LIN {X 0,Y 249.202,Z 538.442,A -85,B 0,C 180,E1 -19004.703,E2 -19004.703} C_VEL
LIN {X 0,Y 249.136,Z 538.448,A -85,B 0,C 180,E1 -19008.077,E2 -19008.077} C_VEL
LIN {X 0,Y 249.084,Z 538.455,A -85,B 0,C 180,E1 -19011.518,E2 -19011.518} C_VEL
LIN {X 0,Y 249.127,Z 538.45,A -85,B 0,C 180,E1 -19015.482,E2 -19015.482} C_VEL
LIN {X 0,Y 249.079,Z 538.459,A -85,B 0,C 180,E1 -19018.993,E2 -19018.993} C_VEL
LIN {X 0,Y 249.032,Z 538.463,A -85,B 0,C 180,E1 -19022.425,E2 -19022.425} C_VEL
LIN {X 0,Y 249.071,Z 538.458,A -85,B 0,C 180,E1 -19026.337,E2 -19026.337} C_VEL
LIN {X 0,Y 249.079,Z 538.453,A -85,B 0,C 180,E1 -19030.463,E2 -19030.463} C_VEL
LIN {X 0,Y 249.089,Z 538.457,A -85,B 0,C 180,E1 -19032.814,E2 -19032.814} C_VEL
LIN {X 0,Y 249.092,Z 538.448,A -85,B 0,C 180,E1 -19037.38,E2 -19037.38} C_VEL
LIN {X 0,Y 249.047,Z 538.461,A -85,B 0,C 180,E1 -19041.624,E2 -19041.624} C_VEL
LIN {X 0,Y 249.055,Z 538.456,A -85,B 0,C 180,E1 -19045.642,E2 -19045.642} C_VEL
LIN {X 0,Y 249.046,Z 538.458,A -85,B 0,C 180,E1 -19049.473,E2 -19049.473} C_VEL
LIN {X 0,Y 249.065,Z 538.462,A -85,B 0,C 180,E1 -19053.162,E2 -19053.162} C_VEL
LIN {X 0,Y 249.055,Z 538.459,A -85,B 0,C 180,E1 -19056.731,E2 -19056.731} C_VEL
LIN {X 0,Y 249.101,Z 538.445,A -85,B 0,C 180,E1 -19060.212,E2 -19060.212} C_VEL
LIN {X 0,Y 249.236,Z 538.437,A -85,B 0,C 180,E1 -19063.622,E2 -19063.622} C_VEL
LIN {X 0,Y 249.247,Z 538.431,A -85,B 0,C 180,E1 -19068.617,E2 -19068.617} C_VEL
LIN {X 0,Y 249.476,Z 538.401,A -85,B 0,C 180,E1 -19071.903,E2 -19071.903} C_VEL
LIN {X 0,Y 249.432,Z 538.412,A -85,B 0,C 180,E1 -19076.77,E2 -19076.77} C_VEL
LIN {X 0,Y 249.73,Z 538.365,A -85,B 0,C 180,E1 -19080.001,E2 -19080.001} C_VEL
LIN {X 0,Y 249.463,Z 538.408,A -85,B 0,C 180,E1 -19083.231,E2 -19083.231} C_VEL
LIN {X 0,Y 249.45,Z 538.405,A -85,B 0,C 180,E1 -19088.099,E2 -19088.099} C_VEL
LIN {X 0,Y 249.218,Z 538.441,A -85,B 0,C 180,E1 -19093.039,E2 -19093.039} C_VEL
LIN {X 0,Y 249.184,Z 538.442,A -85,B 0,C 180,E1 -19094.212,E2 -19094.212} C_VEL
LIN {X 0,Y 248.517,Z 538.528,A -85,B 0,C 180,E1 -19095.561,E2 -19095.561} C_VEL
LIN {X 0,Y 245.6,Z 538.889,A -85,B 0,C 180,E1 -19097.758,E2 -19097.758} C_VEL
LIN {X 0,Y 243.131,Z 539.2,A -85,B 0,C 180,E1 -19099.547,E2 -19099.547} C_VEL
LIN {X 0,Y 242.102,Z 539.328,A -85,B 0,C 180,E1 -19100.938,E2 -19100.938} C_VEL
LIN {X 0,Y 242.035,Z 539.333,A -85,B 0,C 180,E1 -19101.409,E2 -19101.409} C_VEL
LIN {X 0,Y 242.064,Z 539.332,A -85,B 0,C 180,E1 -19105.839,E2 -19105.839} C_VEL
LIN {X 0,Y 242.028,Z 539.335,A -85,B 0,C 180,E1 -19109.581,E2 -19109.581} C_VEL
LIN {X 0,Y 241.989,Z 539.34,A -85,B 0,C 180,E1 -19113.492,E2 -19113.492} C_VEL
LIN {X 0,Y 241.997,Z 539.34,A -85,B 0,C 180,E1 -19117.581,E2 -19117.581} C_VEL
LIN {X 0,Y 241.942,Z 539.347,A -85,B 0,C 180,E1 -19121.922,E2 -19121.922} C_VEL
LIN {X 0,Y 241.991,Z 539.341,A -85,B 0,C 180,E1 -19126.558,E2 -19126.558} C_VEL
LIN {X 0,Y 242.063,Z 539.462,A -85,B 0,C 180,E1 -19131.377,E2 -19131.377} C_VEL
LIN {X 0,Y 244.298,Z 549.492,A -85,B 0,C 180,E1 -19135.282,E2 -19135.282} C_VEL
LIN {X 0,Y 246.378,Z 559.411,A -85,B 0,C 180,E1 -19138.944,E2 -19138.944} C_VEL
LIN {X 0,Y 250.709,Z 571.961,A -85,B 0,C 180,E1 -19139.853,E2 -19139.853} C_VEL
LIN {X 0,Y 255.893,Z 613.107,A -85,B 0,C 180,E1 -19141.765,E2 -19141.765} C_VEL
LIN {X 0,Y 254.09,Z 666.383,A -85,B 0,C 180,E1 -19143.398,E2 -19143.398} C_VEL
LIN {X 0,Y 253.162,Z 679.381,A -85,B 0,C 180,E1 -19144.018,E2 -19144.018} C_VEL
LIN {X 0,Y 251.694,Z 692.993,A -85,B 0,C 180,E1 -19145.019,E2 -19145.019} C_VEL
LIN {X 0,Y 250.086,Z 704.507,A -85,B 0,C 180,E1 -19146.174,E2 -19146.174} C_VEL
LIN {X 0,Y 248.201,Z 716.399,A -85,B 0,C 180,E1 -19147.746,E2 -19147.746} C_VEL
LIN {X 0,Y 246.273,Z 727.047,A -85,B 0,C 180,E1 -19149.539,E2 -19149.539} C_VEL
LIN {X 0,Y 244.509,Z 736.668,A -85,B 0,C 180,E1 -19151.569,E2 -19151.569} C_VEL
LIN {X 0,Y 243.139,Z 744.544,A -85,B 0,C 180,E1 -19153.631,E2 -19153.631} C_VEL
LIN {X 0,Y 241.777,Z 752.217,A -85,B 0,C 180,E1 -19156.125,E2 -19156.125} C_VEL
LIN {X 0,Y 240.683,Z 759.286,A -85,B 0,C 180,E1 -19159.059,E2 -19159.059} C_VEL
LIN {X 0,Y 240.204,Z 763.93,A -85,B 0,C 180,E1 -19161.588,E2 -19161.588} C_VEL
LIN {X 0,Y 240.095,Z 767.755,A -85,B 0,C 180,E1 -19164.414,E2 -19164.414} C_VEL
LIN {X 0,Y 240.067,Z 769.874,A -85,B 0,C 180,E1 -19166.643,E2 -19166.643} C_VEL
LIN {X 0,Y 240.079,Z 770.935,A -85,B 0,C 180,E1 -19168.323,E2 -19168.323} C_VEL
LIN {X 0,Y 240.149,Z 771.574,A -85,B 0,C 180,E1 -19170,E2 -19170} C_VEL
LIN {X 0,Y 240.061,Z 771.798,A -85,B 0,C 180,E1 -19171.678,E2 -19171.678} C_VEL
LIN {X 0,Y 239.982,Z 771.619,A -85,B 0,C 180,E1 -19173.358,E2 -19173.358} C_VEL
LIN {X 0,Y 239.915,Z 770.952,A -85,B 0,C 180,E1 -19175.127,E2 -19175.127} C_VEL
LIN {X 0,Y 240.154,Z 768.543,A -85,B 0,C 180,E1 -19178.414,E2 -19178.414} C_VEL
LIN {X 0,Y 240.703,Z 765.591,A -85,B 0,C 180,E1 -19180.94,E2 -19180.94} C_VEL
LIN {X 0,Y 241.637,Z 761.631,A -85,B 0,C 180,E1 -19183.455,E2 -19183.455} C_VEL
LIN {X 0,Y 243.223,Z 756.564,A -85,B 0,C 180,E1 -19185.932,E2 -19185.932} C_VEL
LIN {X 0,Y 245.134,Z 750.236,A -85,B 0,C 180,E1 -19188.383,E2 -19188.383} C_VEL
LIN {X 0,Y 247.351,Z 742.42,A -85,B 0,C 180,E1 -19190.803,E2 -19190.803} C_VEL
LIN {X 0,Y 250.172,Z 732.673,A -85,B 0,C 180,E1 -19193.159,E2 -19193.159} C_VEL
LIN {X 0,Y 252.937,Z 722.679,A -85,B 0,C 180,E1 -19195.07,E2 -19195.07} C_VEL
LIN {X 0,Y 255.704,Z 711.555,A -85,B 0,C 180,E1 -19196.747,E2 -19196.747} C_VEL
LIN {X 0,Y 258.424,Z 699.033,A -85,B 0,C 180,E1 -19198.198,E2 -19198.198} C_VEL
LIN {X 0,Y 260.641,Z 686.739,A -85,B 0,C 180,E1 -19199.256,E2 -19199.256} C_VEL
LIN {X 0,Y 262.493,Z 673.125,A -85,B 0,C 180,E1 -19200.077,E2 -19200.077} C_VEL
LIN {X 0,Y 263.562,Z 659.455,A -85,B 0,C 180,E1 -19200.616,E2 -19200.616} C_VEL
LIN {X 0,Y 265.646,Z 615.521,A -85,B 0,C 180,E1 -19201.945,E2 -19201.945} C_VEL
LIN {X 0,Y 263.42,Z 595.456,A -85,B 0,C 180,E1 -19203.118,E2 -19203.118} C_VEL
LIN {X 0,Y 261.883,Z 586.129,A -85,B 0,C 180,E1 -19203.783,E2 -19203.783} C_VEL
LIN {X 0,Y 256.187,Z 573.517,A -85,B 0,C 180,E1 -19205.432,E2 -19205.432} C_VEL
LIN {X 0,Y 251.731,Z 564.822,A -85,B 0,C 180,E1 -19206.781,E2 -19206.781} C_VEL
LIN {X 0,Y 249.058,Z 559.92,A -85,B 0,C 180,E1 -19207.624,E2 -19207.624} C_VEL
LIN {X 0,Y 246.628,Z 555.3,A -85,B 0,C 180,E1 -19208.441,E2 -19208.441} C_VEL
LIN {X 0,Y 244.346,Z 546.982,A -85,B 0,C 180,E1 -19212.824,E2 -19212.824} C_VEL
LIN {X 0,Y 242.406,Z 541.046,A -85,B 0,C 180,E1 -19216.452,E2 -19216.452} C_VEL
LIN {X 0,Y 241.976,Z 539.338,A -85,B 0,C 180,E1 -19217.657,E2 -19217.657} C_VEL
LIN {X 0,Y 242,Z 539.336,A -85,B 0,C 180,E1 -19222.419,E2 -19222.419} C_VEL
LIN {X 0,Y 241.989,Z 539.336,A -85,B 0,C 180,E1 -19226.508,E2 -19226.508} C_VEL
LIN {X 0,Y 242.035,Z 539.337,A -85,B 0,C 180,E1 -19230.586,E2 -19230.586} C_VEL
LIN {X 0,Y 242.065,Z 539.333,A -85,B 0,C 180,E1 -19234.182,E2 -19234.182} C_VEL
LIN {X 0,Y 242.05,Z 539.33,A -85,B 0,C 180,E1 -19238.296,E2 -19238.296} C_VEL
LIN {X 0,Y 242.16,Z 539.313,A -85,B 0,C 180,E1 -19243.277,E2 -19243.277} C_VEL
LIN {X 0,Y 242.181,Z 539.318,A -85,B 0,C 180,E1 -19248.279,E2 -19248.279} C_VEL
LIN {X 0,Y 242.422,Z 539.288,A -85,B 0,C 180,E1 -19251.665,E2 -19251.665} C_VEL
LIN {X 0,Y 242.257,Z 539.306,A -85,B 0,C 180,E1 -19255.006,E2 -19255.006} C_VEL
LIN {X 0,Y 242.632,Z 539.26,A -85,B 0,C 180,E1 -19258.339,E2 -19258.339} C_VEL
LIN {X 0,Y 242.634,Z 539.261,A -85,B 0,C 180,E1 -19261.659,E2 -19261.659} C_VEL
LIN {X 0,Y 242.418,Z 539.283,A -85,B 0,C 180,E1 -19266.675,E2 -19266.675} C_VEL
LIN {X 0,Y 242.262,Z 539.308,A -85,B 0,C 180,E1 -19270.023,E2 -19270.023} C_VEL
LIN {X 0,Y 242.181,Z 539.32,A -85,B 0,C 180,E1 -19272.517,E2 -19272.517} C_VEL
LIN {X 0,Y 243.031,Z 541.925,A -85,B 0,C 180,E1 -19272.897,E2 -19272.897} C_VEL
LIN {X 0,Y 244.839,Z 544.043,A -85,B 0,C 180,E1 -19273.486,E2 -19273.486} C_VEL
LIN {X 0,Y 245.625,Z 545.011,A -85,B 0,C 180,E1 -19273.74,E2 -19273.74} C_VEL
LIN {X 0,Y 247.708,Z 548.228,A -85,B 0,C 180,E1 -19274.426,E2 -19274.426} C_VEL
LIN {X 0,Y 249.131,Z 550.181,A -85,B 0,C 180,E1 -19274.864,E2 -19274.864} C_VEL
LIN {X 0,Y 255.936,Z 560.636,A -85,B 0,C 180,E1 -19276.882,E2 -19276.882} C_VEL
LIN {X 0,Y 261.966,Z 571.367,A -85,B 0,C 180,E1 -19278.552,E2 -19278.552} C_VEL
LIN {X 0,Y 266.972,Z 582.249,A -85,B 0,C 180,E1 -19279.921,E2 -19279.921} C_VEL
LIN {X 0,Y 267.197,Z 583.754,A -85,B 0,C 180,E1 -19280.019,E2 -19280.019} C_VEL
LIN {X 0,Y 264.008,Z 643.013,A -85,B 0,C 180,E1 -19281.805,E2 -19281.805} C_VEL
LIN {X 0,Y 262.72,Z 656.866,A -85,B 0,C 180,E1 -19282.537,E2 -19282.537} C_VEL
LIN {X 0,Y 261.055,Z 669.85,A -85,B 0,C 180,E1 -19283.565,E2 -19283.565} C_VEL
LIN {X 0,Y 258.946,Z 682.051,A -85,B 0,C 180,E1 -19284.877,E2 -19284.877} C_VEL
LIN {X 0,Y 256.57,Z 693.258,A -85,B 0,C 180,E1 -19286.43,E2 -19286.43} C_VEL
LIN {X 0,Y 254.034,Z 703.269,A -85,B 0,C 180,E1 -19288.191,E2 -19288.191} C_VEL
LIN {X 0,Y 251.485,Z 712.369,A -85,B 0,C 180,E1 -19290.2,E2 -19290.2} C_VEL
LIN {X 0,Y 248.923,Z 720.553,A -85,B 0,C 180,E1 -19292.441,E2 -19292.441} C_VEL
LIN {X 0,Y 246.775,Z 727.156,A -85,B 0,C 180,E1 -19294.72,E2 -19294.72} C_VEL
LIN {X 0,Y 244.896,Z 732.541,A -85,B 0,C 180,E1 -19297.059,E2 -19297.059} C_VEL
LIN {X 0,Y 243.342,Z 736.838,A -85,B 0,C 180,E1 -19299.447,E2 -19299.447} C_VEL
LIN {X 0,Y 242.128,Z 740.133,A -85,B 0,C 180,E1 -19301.881,E2 -19301.881} C_VEL
LIN {X 0,Y 241.176,Z 742.511,A -85,B 0,C 180,E1 -19304.376,E2 -19304.376} C_VEL
LIN {X 0,Y 240.285,Z 744.252,A -85,B 0,C 180,E1 -19307.724,E2 -19307.724} C_VEL
LIN {X 0,Y 239.976,Z 744.543,A -85,B 0,C 180,E1 -19309.888,E2 -19309.888} C_VEL
LIN {X 0,Y 239.824,Z 744.05,A -85,B 0,C 180,E1 -19312.299,E2 -19312.299} C_VEL
LIN {X 0,Y 239.949,Z 742.461,A -85,B 0,C 180,E1 -19315.094,E2 -19315.094} C_VEL
LIN {X 0,Y 240.48,Z 739.239,A -85,B 0,C 180,E1 -19318.262,E2 -19318.262} C_VEL
LIN {X 0,Y 241.186,Z 735.23,A -85,B 0,C 180,E1 -19320.946,E2 -19320.946} C_VEL
LIN {X 0,Y 242.301,Z 728.97,A -85,B 0,C 180,E1 -19324.046,E2 -19324.046} C_VEL
LIN {X 0,Y 243.655,Z 721.749,A -85,B 0,C 180,E1 -19326.744,E2 -19326.744} C_VEL
LIN {X 0,Y 245.107,Z 714.184,A -85,B 0,C 180,E1 -19328.998,E2 -19328.998} C_VEL
LIN {X 0,Y 246.57,Z 706.345,A -85,B 0,C 180,E1 -19330.91,E2 -19330.91} C_VEL
LIN {X 0,Y 248.345,Z 696.203,A -85,B 0,C 180,E1 -19332.927,E2 -19332.927} C_VEL
LIN {X 0,Y 250.174,Z 684.63,A -85,B 0,C 180,E1 -19334.73,E2 -19334.73} C_VEL
LIN {X 0,Y 251.823,Z 672.374,A -85,B 0,C 180,E1 -19336.221,E2 -19336.221} C_VEL
LIN {X 0,Y 253.139,Z 659.694,A -85,B 0,C 180,E1 -19337.371,E2 -19337.371} C_VEL
LIN {X 0,Y 254.14,Z 646.344,A -85,B 0,C 180,E1 -19338.232,E2 -19338.232} C_VEL
LIN {X 0,Y 254.801,Z 632.802,A -85,B 0,C 180,E1 -19338.767,E2 -19338.767} C_VEL
LIN {X 0,Y 257.003,Z 573.849,A -85,B 0,C 180,E1 -19340.526,E2 -19340.526} C_VEL
LIN {X 0,Y 252.453,Z 562.232,A -85,B 0,C 180,E1 -19341.38,E2 -19341.38} C_VEL
LIN {X 0,Y 243.566,Z 542.387,A -85,B 0,C 180,E1 -19343.042,E2 -19343.042} C_VEL
LIN {X 0,Y 242.401,Z 539.292,A -85,B 0,C 180,E1 -19343.288,E2 -19343.288} C_VEL
LIN {X 0,Y 242.634,Z 539.261,A -85,B 0,C 180,E1 -19348.34,E2 -19348.34} C_VEL
LIN {X 0,Y 242.634,Z 539.261,A -85,B 0,C 180,E1 -19351.66,E2 -19351.66} C_VEL
LIN {X 0,Y 242.432,Z 539.288,A -85,B 0,C 180,E1 -19356.659,E2 -19356.659} C_VEL
LIN {X 0,Y 242.343,Z 539.295,A -85,B 0,C 180,E1 -19360.02,E2 -19360.02} C_VEL
LIN {X 0,Y 242.164,Z 539.32,A -85,B 0,C 180,E1 -19365.141,E2 -19365.141} C_VEL
LIN {X 0,Y 242.07,Z 539.33,A -85,B 0,C 180,E1 -19368.624,E2 -19368.624} C_VEL
LIN {X 0,Y 242.01,Z 539.336,A -85,B 0,C 180,E1 -19372.18,E2 -19372.18} C_VEL
LIN {X 0,Y 242.063,Z 539.328,A -85,B 0,C 180,E1 -19375.838,E2 -19375.838} C_VEL
LIN {X 0,Y 242.026,Z 539.335,A -85,B 0,C 180,E1 -19379.58,E2 -19379.58} C_VEL
LIN {X 0,Y 241.987,Z 539.341,A -85,B 0,C 180,E1 -19383.491,E2 -19383.491} C_VEL
LIN {X 0,Y 242.009,Z 539.334,A -85,B 0,C 180,E1 -19387.577,E2 -19387.577} C_VEL
LIN {X 0,Y 242.032,Z 539.333,A -85,B 0,C 180,E1 -19391.901,E2 -19391.901} C_VEL
LIN {X 0,Y 242.019,Z 539.333,A -85,B 0,C 180,E1 -19396.549,E2 -19396.549} C_VEL
LIN {X 0,Y 242.005,Z 539.334,A -85,B 0,C 180,E1 -19400.292,E2 -19400.292} C_VEL
LIN {X 0,Y 242.031,Z 539.334,A -85,B 0,C 180,E1 -19404.498,E2 -19404.498} C_VEL
LIN {X 0,Y 241.97,Z 539.331,A -85,B 0,C 180,E1 -19408.48,E2 -19408.48} C_VEL
LIN {X 0,Y 242.001,Z 539.337,A -85,B 0,C 180,E1 -19412.313,E2 -19412.313} C_VEL
LIN {X 0,Y 242.035,Z 539.331,A -85,B 0,C 180,E1 -19416.015,E2 -19416.015} C_VEL
LIN {X 0,Y 242.028,Z 539.327,A -85,B 0,C 180,E1 -19419.608,E2 -19419.608} C_VEL
LIN {X 0,Y 242.158,Z 539.321,A -85,B 0,C 180,E1 -19423.279,E2 -19423.279} C_VEL
LIN {X 0,Y 242.18,Z 539.31,A -85,B 0,C 180,E1 -19428.28,E2 -19428.28} C_VEL
LIN {X 0,Y 242.422,Z 539.28,A -85,B 0,C 180,E1 -19431.666,E2 -19431.666} C_VEL
LIN {X 0,Y 242.258,Z 539.306,A -85,B 0,C 180,E1 -19435.008,E2 -19435.008} C_VEL
LIN {X 0,Y 242.632,Z 539.255,A -85,B 0,C 180,E1 -19438.341,E2 -19438.341} C_VEL
LIN {X 0,Y 242.641,Z 539.254,A -85,B 0,C 180,E1 -19441.661,E2 -19441.661} C_VEL
LIN {X 0,Y 242.42,Z 539.285,A -85,B 0,C 180,E1 -19446.66,E2 -19446.66} C_VEL
LIN {X 0,Y 242.263,Z 539.299,A -85,B 0,C 180,E1 -19450.025,E2 -19450.025} C_VEL
LIN {X 0,Y 242.162,Z 539.321,A -85,B 0,C 180,E1 -19455.142,E2 -19455.142} C_VEL
LIN {X 0,Y 242.069,Z 539.327,A -85,B 0,C 180,E1 -19458.625,E2 -19458.625} C_VEL
LIN {X 0,Y 242.035,Z 539.333,A -85,B 0,C 180,E1 -19461.409,E2 -19461.409} C_VEL
LIN {X 0,Y 241.407,Z 539.416,A -85,B 0,C 180,E1 -19462.799,E2 -19462.799} C_VEL
LIN {X 0,Y 238.552,Z 539.776,A -85,B 0,C 180,E1 -19465.065,E2 -19465.065} C_VEL
LIN {X 0,Y 236.094,Z 540.079,A -85,B 0,C 180,E1 -19466.912,E2 -19466.912} C_VEL
LIN {X 0,Y 235.033,Z 540.207,A -85,B 0,C 180,E1 -19468.346,E2 -19468.346} C_VEL
LIN {X 0,Y 234.944,Z 540.216,A -85,B 0,C 180,E1 -19468.832,E2 -19468.832} C_VEL
LIN {X 0,Y 234.948,Z 540.22,A -85,B 0,C 180,E1 -19473.118,E2 -19473.118} C_VEL
LIN {X 0,Y 234.938,Z 540.219,A -85,B 0,C 180,E1 -19476.748,E2 -19476.748} C_VEL
LIN {X 0,Y 234.941,Z 540.22,A -85,B 0,C 180,E1 -19478.946,E2 -19478.946} C_VEL
LIN {X 0,Y 234.922,Z 540.223,A -85,B 0,C 180,E1 -19483.479,E2 -19483.479} C_VEL
LIN {X 0,Y 234.965,Z 540.216,A -85,B 0,C 180,E1 -19486.533,E2 -19486.533} C_VEL
LIN {X 0,Y 235.013,Z 540.33,A -85,B 0,C 180,E1 -19490.776,E2 -19490.776} C_VEL
LIN {X 0,Y 237.181,Z 550.084,A -85,B 0,C 180,E1 -19494.705,E2 -19494.705} C_VEL
LIN {X 0,Y 239.055,Z 558.977,A -85,B 0,C 180,E1 -19498.105,E2 -19498.105} C_VEL
LIN {X 0,Y 244.344,Z 573.596,A -85,B 0,C 180,E1 -19499.238,E2 -19499.238} C_VEL
LIN {X 0,Y 249.409,Z 614.45,A -85,B 0,C 180,E1 -19501.196,E2 -19501.196} C_VEL
LIN {X 0,Y 247.348,Z 668.69,A -85,B 0,C 180,E1 -19502.917,E2 -19502.917} C_VEL
LIN {X 0,Y 246.14,Z 682.575,A -85,B 0,C 180,E1 -19503.676,E2 -19503.676} C_VEL
LIN {X 0,Y 244.638,Z 695.196,A -85,B 0,C 180,E1 -19504.702,E2 -19504.702} C_VEL
LIN {X 0,Y 243.075,Z 706.097,A -85,B 0,C 180,E1 -19505.897,E2 -19505.897} C_VEL
LIN {X 0,Y 241.089,Z 717.567,A -85,B 0,C 180,E1 -19507.505,E2 -19507.505} C_VEL
LIN {X 0,Y 239.187,Z 727.955,A -85,B 0,C 180,E1 -19509.354,E2 -19509.354} C_VEL
LIN {X 0,Y 237.413,Z 737.07,A -85,B 0,C 180,E1 -19511.389,E2 -19511.389} C_VEL
LIN {X 0,Y 235.987,Z 744.978,A -85,B 0,C 180,E1 -19513.566,E2 -19513.566} C_VEL
LIN {X 0,Y 234.624,Z 752.506,A -85,B 0,C 180,E1 -19516.135,E2 -19516.135} C_VEL
LIN {X 0,Y 233.671,Z 758.527,A -85,B 0,C 180,E1 -19518.727,E2 -19518.727} C_VEL
LIN {X 0,Y 233.164,Z 763.256,A -85,B 0,C 180,E1 -19521.332,E2 -19521.332} C_VEL
LIN {X 0,Y 233.032,Z 767.355,A -85,B 0,C 180,E1 -19524.419,E2 -19524.419} C_VEL
LIN {X 0,Y 232.98,Z 769.326,A -85,B 0,C 180,E1 -19526.541,E2 -19526.541} C_VEL
LIN {X 0,Y 233.006,Z 770.449,A -85,B 0,C 180,E1 -19528.272,E2 -19528.272} C_VEL
LIN {X 0,Y 233.071,Z 771.117,A -85,B 0,C 180,E1 -19530,E2 -19530} C_VEL
LIN {X 0,Y 232.985,Z 771.369,A -85,B 0,C 180,E1 -19531.729,E2 -19531.729} C_VEL
LIN {X 0,Y 232.894,Z 771.219,A -85,B 0,C 180,E1 -19533.46,E2 -19533.46} C_VEL
LIN {X 0,Y 232.843,Z 770.655,A -85,B 0,C 180,E1 -19535.195,E2 -19535.195} C_VEL
LIN {X 0,Y 233.098,Z 768.268,A -85,B 0,C 180,E1 -19538.67,E2 -19538.67} C_VEL
LIN {X 0,Y 233.685,Z 765.39,A -85,B 0,C 180,E1 -19541.273,E2 -19541.273} C_VEL
LIN {X 0,Y 234.716,Z 761.502,A -85,B 0,C 180,E1 -19543.859,E2 -19543.859} C_VEL
LIN {X 0,Y 236.374,Z 756.508,A -85,B 0,C 180,E1 -19546.407,E2 -19546.407} C_VEL
LIN {X 0,Y 238.405,Z 750.261,A -85,B 0,C 180,E1 -19548.921,E2 -19548.921} C_VEL
LIN {X 0,Y 240.71,Z 742.57,A -85,B 0,C 180,E1 -19551.405,E2 -19551.405} C_VEL
LIN {X 0,Y 243.163,Z 734.783,A -85,B 0,C 180,E1 -19553.416,E2 -19553.416} C_VEL
LIN {X 0,Y 246.294,Z 724.283,A -85,B 0,C 180,E1 -19555.568,E2 -19555.568} C_VEL
LIN {X 0,Y 249.081,Z 713.685,A -85,B 0,C 180,E1 -19557.29,E2 -19557.29} C_VEL
LIN {X 0,Y 251.9,Z 701.905,A -85,B 0,C 180,E1 -19558.768,E2 -19558.768} C_VEL
LIN {X 0,Y 254.286,Z 689.485,A -85,B 0,C 180,E1 -19559.947,E2 -19559.947} C_VEL
LIN {X 0,Y 256.37,Z 676.585,A -85,B 0,C 180,E1 -19560.816,E2 -19560.816} C_VEL
LIN {X 0,Y 257.709,Z 662.814,A -85,B 0,C 180,E1 -19561.439,E2 -19561.439} C_VEL
LIN {X 0,Y 260.094,Z 616.653,A -85,B 0,C 180,E1 -19562.874,E2 -19562.874} C_VEL
LIN {X 0,Y 258.075,Z 597.538,A -85,B 0,C 180,E1 -19564.04,E2 -19564.04} C_VEL
LIN {X 0,Y 256.781,Z 589.3,A -85,B 0,C 180,E1 -19564.641,E2 -19564.641} C_VEL
LIN {X 0,Y 251.619,Z 577.704,A -85,B 0,C 180,E1 -19566.225,E2 -19566.225} C_VEL
LIN {X 0,Y 247.433,Z 569.349,A -85,B 0,C 180,E1 -19567.566,E2 -19567.566} C_VEL
LIN {X 0,Y 244.395,Z 563.839,A -85,B 0,C 180,E1 -19568.569,E2 -19568.569} C_VEL
LIN {X 0,Y 242.098,Z 559.633,A -85,B 0,C 180,E1 -19569.378,E2 -19569.378} C_VEL
LIN {X 0,Y 239.445,Z 555.129,A -85,B 0,C 180,E1 -19570.332,E2 -19570.332} C_VEL
LIN {X 0,Y 239.177,Z 554.501,A -85,B 0,C 180,E1 -19570.479,E2 -19570.479} C_VEL
LIN {X 0,Y 237.473,Z 548.375,A -85,B 0,C 180,E1 -19573.977,E2 -19573.977} C_VEL
LIN {X 0,Y 235.684,Z 542.635,A -85,B 0,C 180,E1 -19577.718,E2 -19577.718} C_VEL
LIN {X 0,Y 234.92,Z 540.219,A -85,B 0,C 180,E1 -19579.547,E2 -19579.547} C_VEL
LIN {X 0,Y 234.954,Z 540.214,A -85,B 0,C 180,E1 -19583.863,E2 -19583.863} C_VEL
LIN {X 0,Y 234.958,Z 540.219,A -85,B 0,C 180,E1 -19587.424,E2 -19587.424} C_VEL
LIN {X 0,Y 234.949,Z 540.215,A -85,B 0,C 180,E1 -19591.405,E2 -19591.405} C_VEL
LIN {X 0,Y 234.984,Z 540.206,A -85,B 0,C 180,E1 -19595.245,E2 -19595.245} C_VEL
LIN {X 0,Y 235.008,Z 540.203,A -85,B 0,C 180,E1 -19598.969,E2 -19598.969} C_VEL
LIN {X 0,Y 235.093,Z 540.192,A -85,B 0,C 180,E1 -19603.059,E2 -19603.059} C_VEL
LIN {X 0,Y 235.142,Z 540.194,A -85,B 0,C 180,E1 -19607.923,E2 -19607.923} C_VEL
LIN {X 0,Y 235.372,Z 540.163,A -85,B 0,C 180,E1 -19611.413,E2 -19611.413} C_VEL
LIN {X 0,Y 235.399,Z 540.155,A -85,B 0,C 180,E1 -19613.14,E2 -19613.14} C_VEL
LIN {X 0,Y 235.591,Z 540.136,A -85,B 0,C 180,E1 -19618.29,E2 -19618.29} C_VEL
LIN {X 0,Y 235.593,Z 540.138,A -85,B 0,C 180,E1 -19621.709,E2 -19621.709} C_VEL
LIN {X 0,Y 235.369,Z 540.162,A -85,B 0,C 180,E1 -19626.859,E2 -19626.859} C_VEL
LIN {X 0,Y 235.18,Z 540.191,A -85,B 0,C 180,E1 -19630.491,E2 -19630.491} C_VEL
LIN {X 0,Y 236.208,Z 543.144,A -85,B 0,C 180,E1 -19631.008,E2 -19631.008} C_VEL
LIN {X 0,Y 238.689,Z 545.809,A -85,B 0,C 180,E1 -19631.894,E2 -19631.894} C_VEL
LIN {X 0,Y 240.895,Z 549.238,A -85,B 0,C 180,E1 -19632.692,E2 -19632.692} C_VEL
LIN {X 0,Y 242.256,Z 550.995,A -85,B 0,C 180,E1 -19633.152,E2 -19633.152} C_VEL
LIN {X 0,Y 247.457,Z 558.617,A -85,B 0,C 180,E1 -19634.861,E2 -19634.861} C_VEL
LIN {X 0,Y 253.943,Z 569.284,A -85,B 0,C 180,E1 -19636.834,E2 -19636.834} C_VEL
LIN {X 0,Y 258.532,Z 578.029,A -85,B 0,C 180,E1 -19638.159,E2 -19638.159} C_VEL
LIN {X 0,Y 261.583,Z 584.95,A -85,B 0,C 180,E1 -19639.037,E2 -19639.037} C_VEL
LIN {X 0,Y 258.379,Z 643.518,A -85,B 0,C 180,E1 -19640.872,E2 -19640.872} C_VEL
LIN {X 0,Y 257.012,Z 657.282,A -85,B 0,C 180,E1 -19641.611,E2 -19641.611} C_VEL
LIN {X 0,Y 255.251,Z 670.42,A -85,B 0,C 180,E1 -19642.672,E2 -19642.672} C_VEL
LIN {X 0,Y 252.949,Z 683.061,A -85,B 0,C 180,E1 -19644.063,E2 -19644.063} C_VEL
LIN {X 0,Y 250.444,Z 694.164,A -85,B 0,C 180,E1 -19645.645,E2 -19645.645} C_VEL
LIN {X 0,Y 247.741,Z 704.253,A -85,B 0,C 180,E1 -19647.475,E2 -19647.475} C_VEL
LIN {X 0,Y 244.872,Z 713.931,A -85,B 0,C 180,E1 -19649.695,E2 -19649.695} C_VEL
LIN {X 0,Y 242.261,Z 721.749,A -85,B 0,C 180,E1 -19651.951,E2 -19651.951} C_VEL
LIN {X 0,Y 240.028,Z 728.092,A -85,B 0,C 180,E1 -19654.255,E2 -19654.255} C_VEL
LIN {X 0,Y 237.754,Z 734.105,A -85,B 0,C 180,E1 -19657.051,E2 -19657.051} C_VEL
LIN {X 0,Y 235.776,Z 739.204,A -85,B 0,C 180,E1 -19660.269,E2 -19660.269} C_VEL
LIN {X 0,Y 235.13,Z 740.842,A -85,B 0,C 180,E1 -19661.649,E2 -19661.649} C_VEL
LIN {X 0,Y 234.241,Z 742.916,A -85,B 0,C 180,E1 -19663.941,E2 -19663.941} C_VEL
LIN {X 0,Y 233.526,Z 744.262,A -85,B 0,C 180,E1 -19666.242,E2 -19666.242} C_VEL
LIN {X 0,Y 232.982,Z 744.933,A -85,B 0,C 180,E1 -19668.948,E2 -19668.948} C_VEL
LIN {X 0,Y 232.766,Z 744.603,A -85,B 0,C 180,E1 -19671.722,E2 -19671.722} C_VEL
LIN {X 0,Y 232.863,Z 742.884,A -85,B 0,C 180,E1 -19675.011,E2 -19675.011} C_VEL
LIN {X 0,Y 233.411,Z 739.52,A -85,B 0,C 180,E1 -19678.391,E2 -19678.391} C_VEL
LIN {X 0,Y 234.187,Z 735.213,A -85,B 0,C 180,E1 -19681.305,E2 -19681.305} C_VEL
LIN {X 0,Y 235.07,Z 730.446,A -85,B 0,C 180,E1 -19683.754,E2 -19683.754} C_VEL
LIN {X 0,Y 236.228,Z 724.366,A -85,B 0,C 180,E1 -19686.241,E2 -19686.241} C_VEL
LIN {X 0,Y 237.798,Z 716.606,A -85,B 0,C 180,E1 -19688.775,E2 -19688.775} C_VEL
LIN {X 0,Y 239.602,Z 707.289,A -85,B 0,C 180,E1 -19691.177,E2 -19691.177} C_VEL
LIN {X 0,Y 241.274,Z 698.221,A -85,B 0,C 180,E1 -19693.065,E2 -19693.065} C_VEL
LIN {X 0,Y 243.091,Z 687.188,A -85,B 0,C 180,E1 -19694.918,E2 -19694.918} C_VEL
LIN {X 0,Y 244.821,Z 674.908,A -85,B 0,C 180,E1 -19696.512,E2 -19696.512} C_VEL
LIN {X 0,Y 246.255,Z 662.439,A -85,B 0,C 180,E1 -19697.745,E2 -19697.745} C_VEL
LIN {X 0,Y 247.367,Z 649.051,A -85,B 0,C 180,E1 -19698.685,E2 -19698.685} C_VEL
LIN {X 0,Y 248.107,Z 635.587,A -85,B 0,C 180,E1 -19699.287,E2 -19699.287} C_VEL
LIN {X 0,Y 250.412,Z 575.234,A -85,B 0,C 180,E1 -19701.141,E2 -19701.141} C_VEL
LIN {X 0,Y 245.179,Z 562.318,A -85,B 0,C 180,E1 -19702.149,E2 -19702.149} C_VEL
LIN {X 0,Y 236.653,Z 543.491,A -85,B 0,C 180,E1 -19703.807,E2 -19703.807} C_VEL
LIN {X 0,Y 235.404,Z 540.871,A -85,B 0,C 180,E1 -19704.056,E2 -19704.056} C_VEL
LIN {X 0,Y 235.28,Z 540.177,A -85,B 0,C 180,E1 -19704.107,E2 -19704.107} C_VEL
LIN {X 0,Y 235.594,Z 540.138,A -85,B 0,C 180,E1 -19708.291,E2 -19708.291} C_VEL
LIN {X 0,Y 235.594,Z 540.138,A -85,B 0,C 180,E1 -19711.709,E2 -19711.709} C_VEL
LIN {X 0,Y 235.403,Z 540.163,A -85,B 0,C 180,E1 -19716.858,E2 -19716.858} C_VEL
LIN {X 0,Y 235.251,Z 540.179,A -85,B 0,C 180,E1 -19720.326,E2 -19720.326} C_VEL
LIN {X 0,Y 235.111,Z 540.196,A -85,B 0,C 180,E1 -19725.606,E2 -19725.606} C_VEL
LIN {X 0,Y 235.006,Z 540.21,A -85,B 0,C 180,E1 -19729.205,E2 -19729.205} C_VEL
LIN {X 0,Y 234.958,Z 540.216,A -85,B 0,C 180,E1 -19732.883,E2 -19732.883} C_VEL
LIN {X 0,Y 234.966,Z 540.214,A -85,B 0,C 180,E1 -19736.657,E2 -19736.657} C_VEL
LIN {X 0,Y 234.928,Z 540.22,A -85,B 0,C 180,E1 -19740.567,E2 -19740.567} C_VEL
LIN {X 0,Y 234.956,Z 540.217,A -85,B 0,C 180,E1 -19744.633,E2 -19744.633} C_VEL
LIN {X 0,Y 234.962,Z 540.211,A -85,B 0,C 180,E1 -19748.952,E2 -19748.952} C_VEL
LIN {X 0,Y 234.992,Z 540.212,A -85,B 0,C 180,E1 -19753.461,E2 -19753.461} C_VEL
LIN {X 0,Y 234.991,Z 540.209,A -85,B 0,C 180,E1 -19756.539,E2 -19756.539} C_VEL
LIN {X 0,Y 234.95,Z 540.217,A -85,B 0,C 180,E1 -19761.086,E2 -19761.086} C_VEL
LIN {X 0,Y 234.955,Z 540.213,A -85,B 0,C 180,E1 -19765.367,E2 -19765.367} C_VEL
LIN {X 0,Y 234.964,Z 540.21,A -85,B 0,C 180,E1 -19770.158,E2 -19770.158} C_VEL
LIN {X 0,Y 234.989,Z 540.212,A -85,B 0,C 180,E1 -19773.794,E2 -19773.794} C_VEL
LIN {X 0,Y 234.991,Z 540.202,A -85,B 0,C 180,E1 -19778.969,E2 -19778.969} C_VEL
LIN {X 0,Y 235.091,Z 540.199,A -85,B 0,C 180,E1 -19783.06,E2 -19783.06} C_VEL
LIN {X 0,Y 235.112,Z 540.191,A -85,B 0,C 180,E1 -19787.923,E2 -19787.923} C_VEL
LIN {X 0,Y 235.372,Z 540.156,A -85,B 0,C 180,E1 -19791.415,E2 -19791.415} C_VEL
LIN {X 0,Y 235.4,Z 540.157,A -85,B 0,C 180,E1 -19793.142,E2 -19793.142} C_VEL
LIN {X 0,Y 235.591,Z 540.131,A -85,B 0,C 180,E1 -19798.291,E2 -19798.291} C_VEL
LIN {X 0,Y 235.602,Z 540.13,A -85,B 0,C 180,E1 -19801.71,E2 -19801.71} C_VEL
LIN {X 0,Y 235.389,Z 540.161,A -85,B 0,C 180,E1 -19806.86,E2 -19806.86} C_VEL
LIN {X 0,Y 235.21,Z 540.177,A -85,B 0,C 180,E1 -19810.329,E2 -19810.329} C_VEL
LIN {X 0,Y 235.11,Z 540.195,A -85,B 0,C 180,E1 -19815.608,E2 -19815.608} C_VEL
LIN {X 0,Y 235.005,Z 540.21,A -85,B 0,C 180,E1 -19819.207,E2 -19819.207} C_VEL
LIN {X 0,Y 234.958,Z 540.216,A -85,B 0,C 180,E1 -19822.884,E2 -19822.884} C_VEL
LIN {X 0,Y 234.967,Z 540.215,A -85,B 0,C 180,E1 -19826.658,E2 -19826.658} C_VEL
LIN {X 0,Y 234.944,Z 540.216,A -85,B 0,C 180,E1 -19828.832,E2 -19828.832} C_VEL
LIN {X 0,Y 234.266,Z 540.302,A -85,B 0,C 180,E1 -19830.264,E2 -19830.264} C_VEL
LIN {X 0,Y 231.402,Z 540.66,A -85,B 0,C 180,E1 -19832.599,E2 -19832.599} C_VEL
LIN {X 0,Y 228.986,Z 540.96,A -85,B 0,C 180,E1 -19834.503,E2 -19834.503} C_VEL
LIN {X 0,Y 227.969,Z 541.088,A -85,B 0,C 180,E1 -19835.981,E2 -19835.981} C_VEL
LIN {X 0,Y 227.896,Z 541.096,A -85,B 0,C 180,E1 -19836.482,E2 -19836.482} C_VEL
LIN {X 0,Y 227.827,Z 541.103,A -85,B 0,C 180,E1 -19840.377,E2 -19840.377} C_VEL
LIN {X 0,Y 227.85,Z 541.103,A -85,B 0,C 180,E1 -19844.813,E2 -19844.813} C_VEL
LIN {X 0,Y 227.91,Z 541.097,A -85,B 0,C 180,E1 -19847.74,E2 -19847.74} C_VEL
LIN {X 0,Y 227.95,Z 541.133,A -85,B 0,C 180,E1 -19850.117,E2 -19850.117} C_VEL
LIN {X 0,Y 230.063,Z 550.429,A -85,B 0,C 180,E1 -19854.008,E2 -19854.008} C_VEL
LIN {X 0,Y 231.828,Z 558.737,A -85,B 0,C 180,E1 -19857.26,E2 -19857.26} C_VEL
LIN {X 0,Y 238.088,Z 576.073,A -85,B 0,C 180,E1 -19858.644,E2 -19858.644} C_VEL
LIN {X 0,Y 242.905,Z 615.811,A -85,B 0,C 180,E1 -19860.594,E2 -19860.594} C_VEL
LIN {X 0,Y 240.749,Z 667.867,A -85,B 0,C 180,E1 -19862.274,E2 -19862.274} C_VEL
LIN {X 0,Y 239.624,Z 681.334,A -85,B 0,C 180,E1 -19863.02,E2 -19863.02} C_VEL
LIN {X 0,Y 238.079,Z 694.225,A -85,B 0,C 180,E1 -19864.071,E2 -19864.071} C_VEL
LIN {X 0,Y 236.543,Z 704.43,A -85,B 0,C 180,E1 -19865.187,E2 -19865.187} C_VEL
LIN {X 0,Y 234.548,Z 716.147,A -85,B 0,C 180,E1 -19866.842,E2 -19866.842} C_VEL
LIN {X 0,Y 232.493,Z 726.699,A -85,B 0,C 180,E1 -19868.732,E2 -19868.732} C_VEL
LIN {X 0,Y 230.708,Z 735.904,A -85,B 0,C 180,E1 -19870.797,E2 -19870.797} C_VEL
LIN {X 0,Y 229.162,Z 744.036,A -85,B 0,C 180,E1 -19873.062,E2 -19873.062} C_VEL
LIN {X 0,Y 227.721,Z 751.659,A -85,B 0,C 180,E1 -19875.706,E2 -19875.706} C_VEL
LIN {X 0,Y 226.654,Z 757.757,A -85,B 0,C 180,E1 -19878.373,E2 -19878.373} C_VEL
LIN {X 0,Y 226.109,Z 762.564,A -85,B 0,C 180,E1 -19881.06,E2 -19881.06} C_VEL
LIN {X 0,Y 225.919,Z 765.124,A -85,B 0,C 180,E1 -19882.852,E2 -19882.852} C_VEL
LIN {X 0,Y 225.925,Z 767.17,A -85,B 0,C 180,E1 -19884.645,E2 -19884.645} C_VEL
LIN {X 0,Y 225.896,Z 768.771,A -85,B 0,C 180,E1 -19886.433,E2 -19886.433} C_VEL
LIN {X 0,Y 225.934,Z 769.946,A -85,B 0,C 180,E1 -19888.217,E2 -19888.217} C_VEL
LIN {X 0,Y 225.995,Z 770.656,A -85,B 0,C 180,E1 -19890,E2 -19890} C_VEL
LIN {X 0,Y 225.911,Z 770.939,A -85,B 0,C 180,E1 -19891.783,E2 -19891.783} C_VEL
LIN {X 0,Y 225.727,Z 770.455,A -85,B 0,C 180,E1 -19894.91,E2 -19894.91} C_VEL
LIN {X 0,Y 225.825,Z 769.358,A -85,B 0,C 180,E1 -19897.151,E2 -19897.151} C_VEL
LIN {X 0,Y 226.443,Z 766.237,A -85,B 0,C 180,E1 -19900.732,E2 -19900.732} C_VEL
LIN {X 0,Y 227.364,Z 762.758,A -85,B 0,C 180,E1 -19903.405,E2 -19903.405} C_VEL
LIN {X 0,Y 228.935,Z 758.23,A -85,B 0,C 180,E1 -19906.038,E2 -19906.038} C_VEL
LIN {X 0,Y 230.871,Z 752.536,A -85,B 0,C 180,E1 -19908.64,E2 -19908.64} C_VEL
LIN {X 0,Y 233.213,Z 745.492,A -85,B 0,C 180,E1 -19911.2,E2 -19911.2} C_VEL
LIN {X 0,Y 236.153,Z 736.743,A -85,B 0,C 180,E1 -19913.688,E2 -19913.688} C_VEL
LIN {X 0,Y 239.002,Z 727.836,A -85,B 0,C 180,E1 -19915.704,E2 -19915.704} C_VEL
LIN {X 0,Y 242.239,Z 716.946,A -85,B 0,C 180,E1 -19917.658,E2 -19917.658} C_VEL
LIN {X 0,Y 245.016,Z 706.084,A -85,B 0,C 180,E1 -19919.184,E2 -19919.184} C_VEL
LIN {X 0,Y 247.648,Z 694.113,A -85,B 0,C 180,E1 -19920.482,E2 -19920.482} C_VEL
LIN {X 0,Y 249.934,Z 681.778,A -85,B 0,C 180,E1 -19921.463,E2 -19921.463} C_VEL
LIN {X 0,Y 251.606,Z 669.175,A -85,B 0,C 180,E1 -19922.17,E2 -19922.17} C_VEL
LIN {X 0,Y 252.824,Z 651.177,A -85,B 0,C 180,E1 -19922.811,E2 -19922.811} C_VEL
LIN {X 0,Y 254.635,Z 617.858,A -85,B 0,C 180,E1 -19923.857,E2 -19923.857} C_VEL
LIN {X 0,Y 252.821,Z 599.675,A -85,B 0,C 180,E1 -19924.996,E2 -19924.996} C_VEL
LIN {X 0,Y 251.637,Z 592.238,A -85,B 0,C 180,E1 -19925.568,E2 -19925.568} C_VEL
LIN {X 0,Y 246.069,Z 579.457,A -85,B 0,C 180,E1 -19927.415,E2 -19927.415} C_VEL
LIN {X 0,Y 240.631,Z 569.003,A -85,B 0,C 180,E1 -19929.291,E2 -19929.291} C_VEL
LIN {X 0,Y 238.038,Z 564.331,A -85,B 0,C 180,E1 -19930.241,E2 -19930.241} C_VEL
LIN {X 0,Y 234.884,Z 559.07,A -85,B 0,C 180,E1 -19931.435,E2 -19931.435} C_VEL
LIN {X 0,Y 232.184,Z 554.742,A -85,B 0,C 180,E1 -19932.52,E2 -19932.52} C_VEL
LIN {X 0,Y 231.792,Z 553.727,A -85,B 0,C 180,E1 -19932.759,E2 -19932.759} C_VEL
LIN {X 0,Y 229.674,Z 546.844,A -85,B 0,C 180,E1 -19937.255,E2 -19937.255} C_VEL
LIN {X 0,Y 227.893,Z 541.099,A -85,B 0,C 180,E1 -19941.708,E2 -19941.708} C_VEL
LIN {X 0,Y 227.888,Z 541.091,A -85,B 0,C 180,E1 -19946.372,E2 -19946.372} C_VEL
LIN {X 0,Y 227.917,Z 541.095,A -85,B 0,C 180,E1 -19950.437,E2 -19950.437} C_VEL
LIN {X 0,Y 227.926,Z 541.092,A -85,B 0,C 180,E1 -19954.425,E2 -19954.425} C_VEL
LIN {X 0,Y 227.959,Z 541.084,A -85,B 0,C 180,E1 -19958.286,E2 -19958.286} C_VEL
LIN {X 0,Y 228.031,Z 541.071,A -85,B 0,C 180,E1 -19962.825,E2 -19962.825} C_VEL
LIN {X 0,Y 228.089,Z 541.068,A -85,B 0,C 180,E1 -19967.543,E2 -19967.543} C_VEL
LIN {X 0,Y 228.301,Z 541.041,A -85,B 0,C 180,E1 -19971.145,E2 -19971.145} C_VEL
LIN {X 0,Y 228.35,Z 541.035,A -85,B 0,C 180,E1 -19972.928,E2 -19972.928} C_VEL
LIN {X 0,Y 228.55,Z 541.013,A -85,B 0,C 180,E1 -19978.237,E2 -19978.237} C_VEL
LIN {X 0,Y 228.552,Z 541.015,A -85,B 0,C 180,E1 -19981.761,E2 -19981.761} C_VEL
LIN {X 0,Y 228.288,Z 541.047,A -85,B 0,C 180,E1 -19988.241,E2 -19988.241} C_VEL
LIN {X 0,Y 229.214,Z 543.77,A -85,B 0,C 180,E1 -19988.762,E2 -19988.762} C_VEL
LIN {X 0,Y 231.026,Z 545.86,A -85,B 0,C 180,E1 -19989.51,E2 -19989.51} C_VEL
LIN {X 0,Y 231.914,Z 546.79,A -85,B 0,C 180,E1 -19989.859,E2 -19989.859} C_VEL
LIN {X 0,Y 233.865,Z 549.985,A -85,B 0,C 180,E1 -19990.671,E2 -19990.671} C_VEL
LIN {X 0,Y 235.493,Z 551.88,A -85,B 0,C 180,E1 -19991.281,E2 -19991.281} C_VEL
LIN {X 0,Y 238.186,Z 555.592,A -85,B 0,C 180,E1 -19992.27,E2 -19992.27} C_VEL
LIN {X 0,Y 243.757,Z 564.026,A -85,B 0,C 180,E1 -19994.205,E2 -19994.205} C_VEL
LIN {X 0,Y 249.996,Z 574.545,A -85,B 0,C 180,E1 -19996.195,E2 -19996.195} C_VEL
LIN {X 0,Y 254.777,Z 584.062,A -85,B 0,C 180,E1 -19997.663,E2 -19997.663} C_VEL
LIN {X 0,Y 256.165,Z 587.271,A -85,B 0,C 180,E1 -19998.081,E2 -19998.081} C_VEL
LIN {X 0,Y 252.776,Z 644.881,A -85,B 0,C 180,E1 -19999.917,E2 -19999.917} C_VEL
LIN {X 0,Y 251.362,Z 658.305,A -85,B 0,C 180,E1 -20000.664,E2 -20000.664} C_VEL
LIN {X 0,Y 249.61,Z 670.77,A -85,B 0,C 180,E1 -20001.701,E2 -20001.701} C_VEL
LIN {X 0,Y 247.373,Z 682.521,A -85,B 0,C 180,E1 -20003.005,E2 -20003.005} C_VEL
LIN {X 0,Y 244.582,Z 694.251,A -85,B 0,C 180,E1 -20004.68,E2 -20004.68} C_VEL
LIN {X 0,Y 241.744,Z 704.474,A -85,B 0,C 180,E1 -20006.566,E2 -20006.566} C_VEL
LIN {X 0,Y 238.72,Z 714.187,A -85,B 0,C 180,E1 -20008.829,E2 -20008.829} C_VEL
LIN {X 0,Y 235.962,Z 721.957,A -85,B 0,C 180,E1 -20011.099,E2 -20011.099} C_VEL
LIN {X 0,Y 233.63,Z 728.241,A -85,B 0,C 180,E1 -20013.411,E2 -20013.411} C_VEL
LIN {X 0,Y 231.156,Z 734.392,A -85,B 0,C 180,E1 -20016.324,E2 -20016.324} C_VEL
LIN {X 0,Y 229.53,Z 738.304,A -85,B 0,C 180,E1 -20018.74,E2 -20018.74} C_VEL
LIN {X 0,Y 227.777,Z 742.313,A -85,B 0,C 180,E1 -20022.226,E2 -20022.226} C_VEL
LIN {X 0,Y 226.627,Z 744.536,A -85,B 0,C 180,E1 -20025.499,E2 -20025.499} C_VEL
LIN {X 0,Y 226.007,Z 745.339,A -85,B 0,C 180,E1 -20028.27,E2 -20028.27} C_VEL
LIN {X 0,Y 225.698,Z 745.037,A -85,B 0,C 180,E1 -20031.482,E2 -20031.482} C_VEL
LIN {X 0,Y 225.675,Z 743.879,A -85,B 0,C 180,E1 -20034.064,E2 -20034.064} C_VEL
LIN {X 0,Y 226.042,Z 741.403,A -85,B 0,C 180,E1 -20037.083,E2 -20037.083} C_VEL
LIN {X 0,Y 226.795,Z 737.41,A -85,B 0,C 180,E1 -20040.277,E2 -20040.277} C_VEL
LIN {X 0,Y 227.829,Z 731.863,A -85,B 0,C 180,E1 -20043.453,E2 -20043.453} C_VEL
LIN {X 0,Y 229.238,Z 724.723,A -85,B 0,C 180,E1 -20046.513,E2 -20046.513} C_VEL
LIN {X 0,Y 230.775,Z 717.412,A -85,B 0,C 180,E1 -20048.979,E2 -20048.979} C_VEL
LIN {X 0,Y 232.508,Z 708.978,A -85,B 0,C 180,E1 -20051.267,E2 -20051.267} C_VEL
LIN {X 0,Y 234.477,Z 698.39,A -85,B 0,C 180,E1 -20053.561,E2 -20053.561} C_VEL
LIN {X 0,Y 236.267,Z 687.993,A -85,B 0,C 180,E1 -20055.355,E2 -20055.355} C_VEL
LIN {X 0,Y 238.034,Z 675.894,A -85,B 0,C 180,E1 -20056.986,E2 -20056.986} C_VEL
LIN {X 0,Y 239.526,Z 663.532,A -85,B 0,C 180,E1 -20058.255,E2 -20058.255} C_VEL
LIN {X 0,Y 240.637,Z 650.645,A -85,B 0,C 180,E1 -20059.217,E2 -20059.217} C_VEL
LIN {X 0,Y 241.424,Z 637.824,A -85,B 0,C 180,E1 -20059.835,E2 -20059.835} C_VEL
LIN {X 0,Y 243.886,Z 576.818,A -85,B 0,C 180,E1 -20061.768,E2 -20061.768} C_VEL
LIN {X 0,Y 237.938,Z 562.514,A -85,B 0,C 180,E1 -20062.944,E2 -20062.944} C_VEL
LIN {X 0,Y 231.147,Z 547.51,A -85,B 0,C 180,E1 -20064.325,E2 -20064.325} C_VEL
LIN {X 0,Y 228.329,Z 541.848,A -85,B 0,C 180,E1 -20064.896,E2 -20064.896} C_VEL
LIN {X 0,Y 228.197,Z 541.061,A -85,B 0,C 180,E1 -20065.031,E2 -20065.031} C_VEL
LIN {X 0,Y 228.552,Z 541.016,A -85,B 0,C 180,E1 -20068.238,E2 -20068.238} C_VEL
LIN {X 0,Y 228.553,Z 541.015,A -85,B 0,C 180,E1 -20071.762,E2 -20071.762} C_VEL
LIN {X 0,Y 228.356,Z 541.041,A -85,B 0,C 180,E1 -20077.071,E2 -20077.071} C_VEL
LIN {X 0,Y 228.169,Z 541.063,A -85,B 0,C 180,E1 -20080.65,E2 -20080.65} C_VEL
LIN {X 0,Y 228.055,Z 541.074,A -85,B 0,C 180,E1 -20086.102,E2 -20086.102} C_VEL
LIN {X 0,Y 227.939,Z 541.087,A -85,B 0,C 180,E1 -20089.825,E2 -20089.825} C_VEL
LIN {X 0,Y 227.911,Z 541.093,A -85,B 0,C 180,E1 -20093.632,E2 -20093.632} C_VEL
LIN {X 0,Y 227.883,Z 541.098,A -85,B 0,C 180,E1 -20097.555,E2 -20097.555} C_VEL
LIN {X 0,Y 227.869,Z 541.099,A -85,B 0,C 180,E1 -20101.622,E2 -20101.622} C_VEL
LIN {X 0,Y 227.897,Z 541.095,A -85,B 0,C 180,E1 -20105.868,E2 -20105.868} C_VEL
LIN {X 0,Y 227.9,Z 541.09,A -85,B 0,C 180,E1 -20110.36,E2 -20110.36} C_VEL
LIN {X 0,Y 227.915,Z 541.095,A -85,B 0,C 180,E1 -20114.829,E2 -20114.829} C_VEL
LIN {X 0,Y 227.921,Z 541.081,A -85,B 0,C 180,E1 -20117.734,E2 -20117.734} C_VEL
LIN {X 0,Y 227.866,Z 541.098,A -85,B 0,C 180,E1 -20121.915,E2 -20121.915} C_VEL
LIN {X 0,Y 227.885,Z 541.092,A -85,B 0,C 180,E1 -20126.373,E2 -20126.373} C_VEL
LIN {X 0,Y 227.914,Z 541.088,A -85,B 0,C 180,E1 -20130.438,E2 -20130.438} C_VEL
LIN {X 0,Y 227.919,Z 541.093,A -85,B 0,C 180,E1 -20134.426,E2 -20134.426} C_VEL
LIN {X 0,Y 227.942,Z 541.081,A -85,B 0,C 180,E1 -20138.286,E2 -20138.286} C_VEL
LIN {X 0,Y 228.029,Z 541.077,A -85,B 0,C 180,E1 -20142.827,E2 -20142.827} C_VEL
LIN {X 0,Y 228.069,Z 541.069,A -85,B 0,C 180,E1 -20147.544,E2 -20147.544} C_VEL
LIN {X 0,Y 228.301,Z 541.033,A -85,B 0,C 180,E1 -20151.147,E2 -20151.147} C_VEL
LIN {X 0,Y 228.35,Z 541.033,A -85,B 0,C 180,E1 -20152.929,E2 -20152.929} C_VEL
LIN {X 0,Y 228.55,Z 541.008,A -85,B 0,C 180,E1 -20158.239,E2 -20158.239} C_VEL
LIN {X 0,Y 228.561,Z 541.007,A -85,B 0,C 180,E1 -20161.763,E2 -20161.763} C_VEL
LIN {X 0,Y 228.336,Z 541.04,A -85,B 0,C 180,E1 -20167.073,E2 -20167.073} C_VEL
LIN {X 0,Y 228.142,Z 541.058,A -85,B 0,C 180,E1 -20170.652,E2 -20170.652} C_VEL
LIN {X 0,Y 228.06,Z 541.074,A -85,B 0,C 180,E1 -20174.273,E2 -20174.273} C_VEL
LIN {X 0,Y 228,Z 541.079,A -85,B 0,C 180,E1 -20177.954,E2 -20177.954} C_VEL
LIN {X 0,Y 227.927,Z 541.091,A -85,B 0,C 180,E1 -20182.33,E2 -20182.33} C_VEL
LIN {X 0,Y 227.941,Z 541.091,A -85,B 0,C 180,E1 -20186.604,E2 -20186.604} C_VEL
LIN {X 0,Y 227.907,Z 541.093,A -85,B 0,C 180,E1 -20190.297,E2 -20190.297} C_VEL
LIN {X 0,Y 227.888,Z 541.096,A -85,B 0,C 180,E1 -20193.72,E2 -20193.72} C_VEL
LIN {X 0,Y 227.896,Z 541.096,A -85,B 0,C 180,E1 -20196.482,E2 -20196.482} C_VEL
LIN {X 0,Y 227.236,Z 541.179,A -85,B 0,C 180,E1 -20197.956,E2 -20197.956} C_VEL
LIN {X 0,Y 224.329,Z 541.539,A -85,B 0,C 180,E1 -20200.36,E2 -20200.36} C_VEL
LIN {X 0,Y 221.869,Z 541.847,A -85,B 0,C 180,E1 -20202.322,E2 -20202.322} C_VEL
LIN {X 0,Y 220.85,Z 541.975,A -85,B 0,C 180,E1 -20203.848,E2 -20203.848} C_VEL
LIN {X 0,Y 220.786,Z 541.982,A -85,B 0,C 180,E1 -20204.365,E2 -20204.365} C_VEL
LIN {X 0,Y 220.858,Z 541.974,A -85,B 0,C 180,E1 -20208.069,E2 -20208.069} C_VEL
LIN {X 0,Y 220.9,Z 542.027,A -85,B 0,C 180,E1 -20209.467,E2 -20209.467} C_VEL
LIN {X 0,Y 223.102,Z 551.728,A -85,B 0,C 180,E1 -20213.672,E2 -20213.672} C_VEL
LIN {X 0,Y 224.501,Z 558.396,A -85,B 0,C 180,E1 -20216.332,E2 -20216.332} C_VEL
LIN {X 0,Y 231.812,Z 578.097,A -85,B 0,C 180,E1 -20218.004,E2 -20218.004} C_VEL
LIN {X 0,Y 236.317,Z 615.877,A -85,B 0,C 180,E1 -20219.921,E2 -20219.921} C_VEL
LIN {X 0,Y 234.135,Z 667.962,A -85,B 0,C 180,E1 -20221.665,E2 -20221.665} C_VEL
LIN {X 0,Y 232.972,Z 681.259,A -85,B 0,C 180,E1 -20222.428,E2 -20222.428} C_VEL
LIN {X 0,Y 231.383,Z 694.045,A -85,B 0,C 180,E1 -20223.506,E2 -20223.506} C_VEL
LIN {X 0,Y 229.793,Z 704.202,A -85,B 0,C 180,E1 -20224.649,E2 -20224.649} C_VEL
LIN {X 0,Y 227.729,Z 715.881,A -85,B 0,C 180,E1 -20226.348,E2 -20226.348} C_VEL
LIN {X 0,Y 225.612,Z 726.412,A -85,B 0,C 180,E1 -20228.29,E2 -20228.29} C_VEL
LIN {X 0,Y 223.755,Z 735.689,A -85,B 0,C 180,E1 -20230.441,E2 -20230.441} C_VEL
LIN {X 0,Y 222.862,Z 739.988,A -85,B 0,C 180,E1 -20231.618,E2 -20231.618} C_VEL
LIN {X 0,Y 221.486,Z 747.092,A -85,B 0,C 180,E1 -20233.881,E2 -20233.881} C_VEL
LIN {X 0,Y 220.135,Z 754.018,A -85,B 0,C 180,E1 -20236.617,E2 -20236.617} C_VEL
LIN {X 0,Y 219.232,Z 760.369,A -85,B 0,C 180,E1 -20239.845,E2 -20239.845} C_VEL
LIN {X 0,Y 218.846,Z 764.463,A -85,B 0,C 180,E1 -20242.62,E2 -20242.62} C_VEL
LIN {X 0,Y 218.889,Z 766.568,A -85,B 0,C 180,E1 -20244.473,E2 -20244.473} C_VEL
LIN {X 0,Y 218.818,Z 768.202,A -85,B 0,C 180,E1 -20246.317,E2 -20246.317} C_VEL
LIN {X 0,Y 218.864,Z 769.416,A -85,B 0,C 180,E1 -20248.16,E2 -20248.16} C_VEL
LIN {X 0,Y 218.92,Z 770.192,A -85,B 0,C 180,E1 -20250,E2 -20250} C_VEL
LIN {X 0,Y 218.837,Z 770.509,A -85,B 0,C 180,E1 -20251.84,E2 -20251.84} C_VEL
LIN {X 0,Y 218.644,Z 770.168,A -85,B 0,C 180,E1 -20254.82,E2 -20254.82} C_VEL
LIN {X 0,Y 218.754,Z 769.055,A -85,B 0,C 180,E1 -20257.383,E2 -20257.383} C_VEL
LIN {X 0,Y 219.415,Z 766.011,A -85,B 0,C 180,E1 -20261.08,E2 -20261.08} C_VEL
LIN {X 0,Y 220.444,Z 762.621,A -85,B 0,C 180,E1 -20263.834,E2 -20263.834} C_VEL
LIN {X 0,Y 222.107,Z 758.185,A -85,B 0,C 180,E1 -20266.545,E2 -20266.545} C_VEL
LIN {X 0,Y 224.162,Z 752.579,A -85,B 0,C 180,E1 -20269.22,E2 -20269.22} C_VEL
LIN {X 0,Y 226.609,Z 745.635,A -85,B 0,C 180,E1 -20271.849,E2 -20271.849} C_VEL
LIN {X 0,Y 229.669,Z 737.064,A -85,B 0,C 180,E1 -20274.4,E2 -20274.4} C_VEL
LIN {X 0,Y 232.642,Z 728.341,A -85,B 0,C 180,E1 -20276.46,E2 -20276.46} C_VEL
LIN {X 0,Y 236.018,Z 717.682,A -85,B 0,C 180,E1 -20278.452,E2 -20278.452} C_VEL
LIN {X 0,Y 238.887,Z 707.192,A -85,B 0,C 180,E1 -20280.008,E2 -20280.008} C_VEL
LIN {X 0,Y 241.618,Z 695.674,A -85,B 0,C 180,E1 -20281.327,E2 -20281.327} C_VEL
LIN {X 0,Y 243.961,Z 683.921,A -85,B 0,C 180,E1 -20282.326,E2 -20282.326} C_VEL
LIN {X 0,Y 246.018,Z 670.081,A -85,B 0,C 180,E1 -20283.161,E2 -20283.161} C_VEL
LIN {X 0,Y 247.164,Z 654.968,A -85,B 0,C 180,E1 -20283.746,E2 -20283.746} C_VEL
LIN {X 0,Y 249.214,Z 618.454,A -85,B 0,C 180,E1 -20284.918,E2 -20284.918} C_VEL
LIN {X 0,Y 247.583,Z 601.005,A -85,B 0,C 180,E1 -20286.062,E2 -20286.062} C_VEL
LIN {X 0,Y 246.696,Z 595.401,A -85,B 0,C 180,E1 -20286.521,E2 -20286.521} C_VEL
LIN {X 0,Y 241.572,Z 583.526,A -85,B 0,C 180,E1 -20288.311,E2 -20288.311} C_VEL
LIN {X 0,Y 236.411,Z 573.299,A -85,B 0,C 180,E1 -20290.224,E2 -20290.224} C_VEL
LIN {X 0,Y 233.867,Z 568.772,A -85,B 0,C 180,E1 -20291.199,E2 -20291.199} C_VEL
LIN {X 0,Y 231.363,Z 564.389,A -85,B 0,C 180,E1 -20292.223,E2 -20292.223} C_VEL
LIN {X 0,Y 227.808,Z 558.623,A -85,B 0,C 180,E1 -20293.742,E2 -20293.742} C_VEL
LIN {X 0,Y 224.764,Z 554.03,A -85,B 0,C 180,E1 -20295.131,E2 -20295.131} C_VEL
LIN {X 0,Y 224.271,Z 552.857,A -85,B 0,C 180,E1 -20295.479,E2 -20295.479} C_VEL
LIN {X 0,Y 222.642,Z 547.721,A -85,B 0,C 180,E1 -20299.251,E2 -20299.251} C_VEL
LIN {X 0,Y 221.345,Z 543.859,A -85,B 0,C 180,E1 -20302.539,E2 -20302.539} C_VEL
LIN {X 0,Y 220.838,Z 541.976,A -85,B 0,C 180,E1 -20304.353,E2 -20304.353} C_VEL
LIN {X 0,Y 220.867,Z 541.966,A -85,B 0,C 180,E1 -20309.394,E2 -20309.394} C_VEL
LIN {X 0,Y 220.893,Z 541.967,A -85,B 0,C 180,E1 -20313.548,E2 -20313.548} C_VEL
LIN {X 0,Y 220.875,Z 541.972,A -85,B 0,C 180,E1 -20317.552,E2 -20317.552} C_VEL
LIN {X 0,Y 220.981,Z 541.95,A -85,B 0,C 180,E1 -20322.57,E2 -20322.57} C_VEL
LIN {X 0,Y 221.022,Z 541.945,A -85,B 0,C 180,E1 -20327.138,E2 -20327.138} C_VEL
LIN {X 0,Y 221.232,Z 541.919,A -85,B 0,C 180,E1 -20330.86,E2 -20330.86} C_VEL
LIN {X 0,Y 221.301,Z 541.914,A -85,B 0,C 180,E1 -20332.701,E2 -20332.701} C_VEL
LIN {X 0,Y 221.508,Z 541.889,A -85,B 0,C 180,E1 -20338.181,E2 -20338.181} C_VEL
LIN {X 0,Y 221.51,Z 541.893,A -85,B 0,C 180,E1 -20341.817,E2 -20341.817} C_VEL
LIN {X 0,Y 221.151,Z 541.978,A -85,B 0,C 180,E1 -20345.527,E2 -20345.527} C_VEL
LIN {X 0,Y 222.027,Z 544.515,A -85,B 0,C 180,E1 -20346.075,E2 -20346.075} C_VEL
LIN {X 0,Y 223.928,Z 546.604,A -85,B 0,C 180,E1 -20346.985,E2 -20346.985} C_VEL
LIN {X 0,Y 225.259,Z 547.675,A -85,B 0,C 180,E1 -20347.571,E2 -20347.571} C_VEL
LIN {X 0,Y 227.079,Z 550.793,A -85,B 0,C 180,E1 -20348.448,E2 -20348.448} C_VEL
LIN {X 0,Y 228.855,Z 552.867,A -85,B 0,C 180,E1 -20349.2,E2 -20349.2} C_VEL
LIN {X 0,Y 231.42,Z 556.494,A -85,B 0,C 180,E1 -20350.266,E2 -20350.266} C_VEL
LIN {X 0,Y 235.95,Z 563.091,A -85,B 0,C 180,E1 -20352.034,E2 -20352.034} C_VEL
LIN {X 0,Y 239.909,Z 569.127,A -85,B 0,C 180,E1 -20353.452,E2 -20353.452} C_VEL
LIN {X 0,Y 245.759,Z 579.197,A -85,B 0,C 180,E1 -20355.433,E2 -20355.433} C_VEL
LIN {X 0,Y 250.112,Z 587.935,A -85,B 0,C 180,E1 -20356.833,E2 -20356.833} C_VEL
LIN {X 0,Y 250.808,Z 589.708,A -85,B 0,C 180,E1 -20357.067,E2 -20357.067} C_VEL
LIN {X 0,Y 247.353,Z 645.303,A -85,B 0,C 180,E1 -20358.881,E2 -20358.881} C_VEL
LIN {X 0,Y 245.861,Z 658.833,A -85,B 0,C 180,E1 -20359.644,E2 -20359.644} C_VEL
LIN {X 0,Y 243.928,Z 671.688,A -85,B 0,C 180,E1 -20360.735,E2 -20360.735} C_VEL
LIN {X 0,Y 241.536,Z 683.603,A -85,B 0,C 180,E1 -20362.094,E2 -20362.094} C_VEL
LIN {X 0,Y 238.712,Z 694.899,A -85,B 0,C 180,E1 -20363.749,E2 -20363.749} C_VEL
LIN {X 0,Y 235.782,Z 704.877,A -85,B 0,C 180,E1 -20365.625,E2 -20365.625} C_VEL
LIN {X 0,Y 232.614,Z 714.466,A -85,B 0,C 180,E1 -20367.906,E2 -20367.906} C_VEL
LIN {X 0,Y 229.732,Z 722.182,A -85,B 0,C 180,E1 -20370.208,E2 -20370.208} C_VEL
LIN {X 0,Y 227.422,Z 727.982,A -85,B 0,C 180,E1 -20372.361,E2 -20372.361} C_VEL
LIN {X 0,Y 225.231,Z 733.304,A -85,B 0,C 180,E1 -20374.813,E2 -20374.813} C_VEL
LIN {X 0,Y 222.896,Z 738.554,A -85,B 0,C 180,E1 -20377.979,E2 -20377.979} C_VEL
LIN {X 0,Y 221.523,Z 741.521,A -85,B 0,C 180,E1 -20380.412,E2 -20380.412} C_VEL
LIN {X 0,Y 220.426,Z 743.637,A -85,B 0,C 180,E1 -20382.836,E2 -20382.836} C_VEL
LIN {X 0,Y 219.61,Z 745.028,A -85,B 0,C 180,E1 -20385.249,E2 -20385.249} C_VEL
LIN {X 0,Y 219.027,Z 745.726,A -85,B 0,C 180,E1 -20387.637,E2 -20387.637} C_VEL
LIN {X 0,Y 218.645,Z 745.656,A -85,B 0,C 180,E1 -20390.482,E2 -20390.482} C_VEL
LIN {X 0,Y 218.556,Z 744.552,A -85,B 0,C 180,E1 -20393.504,E2 -20393.504} C_VEL
LIN {X 0,Y 218.915,Z 741.949,A -85,B 0,C 180,E1 -20396.924,E2 -20396.924} C_VEL
LIN {X 0,Y 219.558,Z 738.597,A -85,B 0,C 180,E1 -20399.797,E2 -20399.797} C_VEL
LIN {X 0,Y 220.576,Z 733.198,A -85,B 0,C 180,E1 -20403.141,E2 -20403.141} C_VEL
LIN {X 0,Y 221.929,Z 726.623,A -85,B 0,C 180,E1 -20406.187,E2 -20406.187} C_VEL
LIN {X 0,Y 223.493,Z 719.419,A -85,B 0,C 180,E1 -20408.8,E2 -20408.8} C_VEL
LIN {X 0,Y 225.358,Z 710.61,A -85,B 0,C 180,E1 -20411.358,E2 -20411.358} C_VEL
LIN {X 0,Y 227.204,Z 701.36,A -85,B 0,C 180,E1 -20413.514,E2 -20413.514} C_VEL
LIN {X 0,Y 229.212,Z 690.213,A -85,B 0,C 180,E1 -20415.575,E2 -20415.575} C_VEL
LIN {X 0,Y 230.983,Z 679.036,A -85,B 0,C 180,E1 -20417.208,E2 -20417.208} C_VEL
LIN {X 0,Y 232.564,Z 666.998,A -85,B 0,C 180,E1 -20418.562,E2 -20418.562} C_VEL
LIN {X 0,Y 233.864,Z 653.411,A -85,B 0,C 180,E1 -20419.681,E2 -20419.681} C_VEL
LIN {X 0,Y 234.788,Z 639.946,A -85,B 0,C 180,E1 -20420.406,E2 -20420.406} C_VEL
LIN {X 0,Y 237.377,Z 578.361,A -85,B 0,C 180,E1 -20422.419,E2 -20422.419} C_VEL
LIN {X 0,Y 227.424,Z 555.163,A -85,B 0,C 180,E1 -20424.488,E2 -20424.488} C_VEL
LIN {X 0,Y 221.392,Z 542.969,A -85,B 0,C 180,E1 -20425.761,E2 -20425.761} C_VEL
LIN {X 0,Y 221.169,Z 541.934,A -85,B 0,C 180,E1 -20425.9,E2 -20425.9} C_VEL
LIN {X 0,Y 221.51,Z 541.893,A -85,B 0,C 180,E1 -20428.182,E2 -20428.182} C_VEL
LIN {X 0,Y 221.511,Z 541.893,A -85,B 0,C 180,E1 -20431.818,E2 -20431.818} C_VEL
LIN {X 0,Y 221.309,Z 541.918,A -85,B 0,C 180,E1 -20437.298,E2 -20437.298} C_VEL
LIN {X 0,Y 221.114,Z 541.941,A -85,B 0,C 180,E1 -20440.994,E2 -20440.994} C_VEL
LIN {X 0,Y 221.013,Z 541.953,A -85,B 0,C 180,E1 -20446.63,E2 -20446.63} C_VEL
LIN {X 0,Y 220.889,Z 541.966,A -85,B 0,C 180,E1 -20450.486,E2 -20450.486} C_VEL
LIN {X 0,Y 220.864,Z 541.971,A -85,B 0,C 180,E1 -20454.435,E2 -20454.435} C_VEL
LIN {X 0,Y 220.833,Z 541.976,A -85,B 0,C 180,E1 -20458.513,E2 -20458.513} C_VEL
LIN {X 0,Y 220.82,Z 541.979,A -85,B 0,C 180,E1 -20462.755,E2 -20462.755} C_VEL
LIN {X 0,Y 220.834,Z 541.972,A -85,B 0,C 180,E1 -20467.288,E2 -20467.288} C_VEL
LIN {X 0,Y 220.869,Z 541.97,A -85,B 0,C 180,E1 -20471.928,E2 -20471.928} C_VEL
LIN {X 0,Y 220.869,Z 541.967,A -85,B 0,C 180,E1 -20475.572,E2 -20475.572} C_VEL
LIN {X 0,Y 220.853,Z 541.968,A -85,B 0,C 180,E1 -20479.792,E2 -20479.792} C_VEL
LIN {X 0,Y 220.83,Z 541.977,A -85,B 0,C 180,E1 -20482.795,E2 -20482.795} C_VEL
LIN {X 0,Y 220.819,Z 541.966,A -85,B 0,C 180,E1 -20487.245,E2 -20487.245} C_VEL
LIN {X 0,Y 220.831,Z 541.976,A -85,B 0,C 180,E1 -20491.487,E2 -20491.487} C_VEL
LIN {X 0,Y 220.857,Z 541.971,A -85,B 0,C 180,E1 -20495.565,E2 -20495.565} C_VEL
LIN {X 0,Y 220.878,Z 541.958,A -85,B 0,C 180,E1 -20499.514,E2 -20499.514} C_VEL
LIN {X 0,Y 221.01,Z 541.954,A -85,B 0,C 180,E1 -20503.371,E2 -20503.371} C_VEL
LIN {X 0,Y 221.101,Z 541.932,A -85,B 0,C 180,E1 -20509.006,E2 -20509.006} C_VEL
LIN {X 0,Y 221.285,Z 541.912,A -85,B 0,C 180,E1 -20512.702,E2 -20512.702} C_VEL
LIN {X 0,Y 221.508,Z 541.885,A -85,B 0,C 180,E1 -20518.183,E2 -20518.183} C_VEL
LIN {X 0,Y 221.519,Z 541.883,A -85,B 0,C 180,E1 -20521.819,E2 -20521.819} C_VEL
LIN {X 0,Y 221.268,Z 541.918,A -85,B 0,C 180,E1 -20527.3,E2 -20527.3} C_VEL
LIN {X 0,Y 221.063,Z 541.941,A -85,B 0,C 180,E1 -20530.997,E2 -20530.997} C_VEL
LIN {X 0,Y 220.992,Z 541.956,A -85,B 0,C 180,E1 -20534.74,E2 -20534.74} C_VEL
LIN {X 0,Y 220.919,Z 541.96,A -85,B 0,C 180,E1 -20538.551,E2 -20538.551} C_VEL
LIN {X 0,Y 220.893,Z 541.968,A -85,B 0,C 180,E1 -20542.684,E2 -20542.684} C_VEL
LIN {X 0,Y 220.884,Z 541.972,A -85,B 0,C 180,E1 -20547.017,E2 -20547.017} C_VEL
LIN {X 0,Y 220.862,Z 541.971,A -85,B 0,C 180,E1 -20550.78,E2 -20550.78} C_VEL
LIN {X 0,Y 220.813,Z 541.977,A -85,B 0,C 180,E1 -20554.954,E2 -20554.954} C_VEL
LIN {X 0,Y 220.838,Z 541.976,A -85,B 0,C 180,E1 -20557.289,E2 -20557.289} C_VEL
LIN {X 0,Y 220.794,Z 541.982,A -85,B 0,C 180,E1 -20561.948,E2 -20561.948} C_VEL
LIN {X 0,Y 220.786,Z 541.982,A -85,B 0,C 180,E1 -20564.365,E2 -20564.365} C_VEL
LIN {X 0,Y 220.104,Z 542.072,A -85,B 0,C 180,E1 -20565.413,E2 -20565.413} C_VEL
LIN {X 0,Y 217.191,Z 542.432,A -85,B 0,C 180,E1 -20567.065,E2 -20567.065} C_VEL
LIN {X 0,Y 214.572,Z 543.37,A -85,B 0,C 180,E1 -20568.691,E2 -20568.691} C_VEL
LIN {X 0,Y 214.247,Z 544.66,A -85,B 0,C 180,E1 -20569.581,E2 -20569.581} C_VEL
LIN {X 0,Y 214.286,Z 544.817,A -85,B 0,C 180,E1 -20569.657,E2 -20569.657} C_VEL
LIN {X 0,Y 216.297,Z 553.755,A -85,B 0,C 180,E1 -20573.633,E2 -20573.633} C_VEL
LIN {X 0,Y 217.117,Z 557.727,A -85,B 0,C 180,E1 -20575.325,E2 -20575.325} C_VEL
LIN {X 0,Y 225.479,Z 579.905,A -85,B 0,C 180,E1 -20577.308,E2 -20577.308} C_VEL
LIN {X 0,Y 229.806,Z 616.776,A -85,B 0,C 180,E1 -20579.248,E2 -20579.248} C_VEL
LIN {X 0,Y 227.55,Z 668.046,A -85,B 0,C 180,E1 -20581.02,E2 -20581.02} C_VEL
LIN {X 0,Y 226.347,Z 681.179,A -85,B 0,C 180,E1 -20581.802,E2 -20581.802} C_VEL
LIN {X 0,Y 224.711,Z 693.859,A -85,B 0,C 180,E1 -20582.907,E2 -20582.907} C_VEL
LIN {X 0,Y 223.073,Z 703.973,A -85,B 0,C 180,E1 -20584.079,E2 -20584.079} C_VEL
LIN {X 0,Y 220.92,Z 715.614,A -85,B 0,C 180,E1 -20585.822,E2 -20585.822} C_VEL
LIN {X 0,Y 218.75,Z 726.126,A -85,B 0,C 180,E1 -20587.821,E2 -20587.821} C_VEL
LIN {X 0,Y 216.805,Z 735.484,A -85,B 0,C 180,E1 -20590.066,E2 -20590.066} C_VEL
LIN {X 0,Y 215.785,Z 740.431,A -85,B 0,C 180,E1 -20591.486,E2 -20591.486} C_VEL
LIN {X 0,Y 214.134,Z 748.645,A -85,B 0,C 180,E1 -20594.29,E2 -20594.29} C_VEL
LIN {X 0,Y 212.98,Z 754.184,A -85,B 0,C 180,E1 -20596.645,E2 -20596.645} C_VEL
LIN {X 0,Y 212.192,Z 759.6,A -85,B 0,C 180,E1 -20599.504,E2 -20599.504} C_VEL
LIN {X 0,Y 211.8,Z 763.782,A -85,B 0,C 180,E1 -20602.373,E2 -20602.373} C_VEL
LIN {X 0,Y 211.797,Z 766.218,A -85,B 0,C 180,E1 -20604.561,E2 -20604.561} C_VEL
LIN {X 0,Y 211.794,Z 768.883,A -85,B 0,C 180,E1 -20608.098,E2 -20608.098} C_VEL
LIN {X 0,Y 211.848,Z 769.714,A -85,B 0,C 180,E1 -20610,E2 -20610} C_VEL
LIN {X 0,Y 211.763,Z 770.078,A -85,B 0,C 180,E1 -20611.902,E2 -20611.902} C_VEL
LIN {X 0,Y 211.567,Z 769.877,A -85,B 0,C 180,E1 -20614.74,E2 -20614.74} C_VEL
LIN {X 0,Y 211.675,Z 768.743,A -85,B 0,C 180,E1 -20617.632,E2 -20617.632} C_VEL
LIN {X 0,Y 211.945,Z 767.484,A -85,B 0,C 180,E1 -20619.543,E2 -20619.543} C_VEL
LIN {X 0,Y 212.726,Z 764.832,A -85,B 0,C 180,E1 -20622.4,E2 -20622.4} C_VEL
LIN {X 0,Y 214.06,Z 761.184,A -85,B 0,C 180,E1 -20625.227,E2 -20625.227} C_VEL
LIN {X 0,Y 215.905,Z 756.459,A -85,B 0,C 180,E1 -20628.013,E2 -20628.013} C_VEL
LIN {X 0,Y 218.318,Z 750.541,A -85,B 0,C 180,E1 -20630.738,E2 -20630.738} C_VEL
LIN {X 0,Y 221.029,Z 743.222,A -85,B 0,C 180,E1 -20633.419,E2 -20633.419} C_VEL
LIN {X 0,Y 224.448,Z 734.2,A -85,B 0,C 180,E1 -20635.999,E2 -20635.999} C_VEL
LIN {X 0,Y 227.678,Z 725.004,A -85,B 0,C 180,E1 -20638.082,E2 -20638.082} C_VEL
LIN {X 0,Y 230.883,Z 714.879,A -85,B 0,C 180,E1 -20639.897,E2 -20639.897} C_VEL
LIN {X 0,Y 234.043,Z 703.744,A -85,B 0,C 180,E1 -20641.449,E2 -20641.449} C_VEL
LIN {X 0,Y 236.924,Z 691.425,A -85,B 0,C 180,E1 -20642.775,E2 -20642.775} C_VEL
LIN {X 0,Y 239.436,Z 678.383,A -85,B 0,C 180,E1 -20643.769,E2 -20643.769} C_VEL
LIN {X 0,Y 241.181,Z 664.779,A -85,B 0,C 180,E1 -20644.492,E2 -20644.492} C_VEL
LIN {X 0,Y 244.007,Z 619.356,A -85,B 0,C 180,E1 -20646.02,E2 -20646.02} C_VEL
LIN {X 0,Y 242.445,Z 602.119,A -85,B 0,C 180,E1 -20647.194,E2 -20647.194} C_VEL
LIN {X 0,Y 241.851,Z 598.561,A -85,B 0,C 180,E1 -20647.508,E2 -20647.508} C_VEL
LIN {X 0,Y 237.059,Z 587.29,A -85,B 0,C 180,E1 -20649.309,E2 -20649.309} C_VEL
LIN {X 0,Y 232.339,Z 577.722,A -85,B 0,C 180,E1 -20651.158,E2 -20651.158} C_VEL
LIN {X 0,Y 228.096,Z 569.969,A -85,B 0,C 180,E1 -20652.96,E2 -20652.96} C_VEL
LIN {X 0,Y 224.487,Z 564.047,A -85,B 0,C 180,E1 -20654.582,E2 -20654.582} C_VEL
LIN {X 0,Y 220.721,Z 558.151,A -85,B 0,C 180,E1 -20656.44,E2 -20656.44} C_VEL
LIN {X 0,Y 217.233,Z 553.107,A -85,B 0,C 180,E1 -20658.315,E2 -20658.315} C_VEL
LIN {X 0,Y 216.748,Z 552.072,A -85,B 0,C 180,E1 -20658.643,E2 -20658.643} C_VEL
LIN {X 0,Y 215.659,Z 548.368,A -85,B 0,C 180,E1 -20661.742,E2 -20661.742} C_VEL
LIN {X 0,Y 214.438,Z 545.046,A -85,B 0,C 180,E1 -20665.018,E2 -20665.018} C_VEL
LIN {X 0,Y 213.788,Z 542.855,A -85,B 0,C 180,E1 -20667.71,E2 -20667.71} C_VEL
LIN {X 0,Y 213.824,Z 542.842,A -85,B 0,C 180,E1 -20672.602,E2 -20672.602} C_VEL
LIN {X 0,Y 213.85,Z 542.843,A -85,B 0,C 180,E1 -20676.952,E2 -20676.952} C_VEL
LIN {X 0,Y 213.929,Z 542.829,A -85,B 0,C 180,E1 -20682.304,E2 -20682.304} C_VEL
LIN {X 0,Y 213.976,Z 542.821,A -85,B 0,C 180,E1 -20686.707,E2 -20686.707} C_VEL
LIN {X 0,Y 214.163,Z 542.798,A -85,B 0,C 180,E1 -20690.555,E2 -20690.555} C_VEL
LIN {X 0,Y 214.236,Z 542.796,A -85,B 0,C 180,E1 -20692.459,E2 -20692.459} C_VEL
LIN {X 0,Y 214.442,Z 542.768,A -85,B 0,C 180,E1 -20698.121,E2 -20698.121} C_VEL
LIN {X 0,Y 214.55,Z 542.753,A -85,B 0,C 180,E1 -20699.999,E2 -20699.999} C_VEL
LIN {X 0,Y 214.342,Z 542.785,A -85,B 0,C 180,E1 -20702.348,E2 -20702.348} C_VEL
LIN {X 0,Y 215.044,Z 545.275,A -85,B 0,C 180,E1 -20702.926,E2 -20702.926} C_VEL
LIN {X 0,Y 216.747,Z 547.474,A -85,B 0,C 180,E1 -20703.95,E2 -20703.95} C_VEL
LIN {X 0,Y 218.446,Z 548.728,A -85,B 0,C 180,E1 -20704.841,E2 -20704.841} C_VEL
LIN {X 0,Y 220.222,Z 551.741,A -85,B 0,C 180,E1 -20705.838,E2 -20705.838} C_VEL
LIN {X 0,Y 222.487,Z 553.973,A -85,B 0,C 180,E1 -20706.916,E2 -20706.916} C_VEL
LIN {X 0,Y 224.899,Z 557.544,A -85,B 0,C 180,E1 -20708.083,E2 -20708.083} C_VEL
LIN {X 0,Y 226.375,Z 559.686,A -85,B 0,C 180,E1 -20708.76,E2 -20708.76} C_VEL
LIN {X 0,Y 229.658,Z 564.307,A -85,B 0,C 180,E1 -20710.151,E2 -20710.151} C_VEL
LIN {X 0,Y 234.7,Z 571.859,A -85,B 0,C 180,E1 -20712.149,E2 -20712.149} C_VEL
LIN {X 0,Y 240.937,Z 582.572,A -85,B 0,C 180,E1 -20714.409,E2 -20714.409} C_VEL
LIN {X 0,Y 245.265,Z 591.348,A -85,B 0,C 180,E1 -20715.893,E2 -20715.893} C_VEL
LIN {X 0,Y 245.603,Z 592.161,A -85,B 0,C 180,E1 -20716.01,E2 -20716.01} C_VEL
LIN {X 0,Y 242.083,Z 645.638,A -85,B 0,C 180,E1 -20717.773,E2 -20717.773} C_VEL
LIN {X 0,Y 240.563,Z 658.809,A -85,B 0,C 180,E1 -20718.523,E2 -20718.523} C_VEL
LIN {X 0,Y 238.666,Z 671.091,A -85,B 0,C 180,E1 -20719.561,E2 -20719.561} C_VEL
LIN {X 0,Y 236.189,Z 683.023,A -85,B 0,C 180,E1 -20720.919,E2 -20720.919} C_VEL
LIN {X 0,Y 233.236,Z 694.265,A -85,B 0,C 180,E1 -20722.555,E2 -20722.555} C_VEL
LIN {X 0,Y 230.208,Z 704.395,A -85,B 0,C 180,E1 -20724.444,E2 -20724.444} C_VEL
LIN {X 0,Y 226.81,Z 714.18,A -85,B 0,C 180,E1 -20726.771,E2 -20726.771} C_VEL
LIN {X 0,Y 223.715,Z 722.105,A -85,B 0,C 180,E1 -20729.146,E2 -20729.146} C_VEL
LIN {X 0,Y 220.994,Z 728.544,A -85,B 0,C 180,E1 -20731.573,E2 -20731.573} C_VEL
LIN {X 0,Y 218.194,Z 734.806,A -85,B 0,C 180,E1 -20734.625,E2 -20734.625} C_VEL
LIN {X 0,Y 216.268,Z 738.853,A -85,B 0,C 180,E1 -20737.205,E2 -20737.205} C_VEL
LIN {X 0,Y 214.769,Z 741.867,A -85,B 0,C 180,E1 -20739.737,E2 -20739.737} C_VEL
LIN {X 0,Y 213.087,Z 744.807,A -85,B 0,C 180,E1 -20743.483,E2 -20743.483} C_VEL
LIN {X 0,Y 212.128,Z 746.053,A -85,B 0,C 180,E1 -20746.791,E2 -20746.791} C_VEL
LIN {X 0,Y 211.606,Z 746.133,A -85,B 0,C 180,E1 -20749.807,E2 -20749.807} C_VEL
LIN {X 0,Y 211.488,Z 745.003,A -85,B 0,C 180,E1 -20753.263,E2 -20753.263} C_VEL
LIN {X 0,Y 211.681,Z 743.057,A -85,B 0,C 180,E1 -20756.099,E2 -20756.099} C_VEL
LIN {X 0,Y 212.352,Z 739.641,A -85,B 0,C 180,E1 -20759.37,E2 -20759.37} C_VEL
LIN {X 0,Y 213.357,Z 734.502,A -85,B 0,C 180,E1 -20762.793,E2 -20762.793} C_VEL
LIN {X 0,Y 214.516,Z 728.936,A -85,B 0,C 180,E1 -20765.613,E2 -20765.613} C_VEL
LIN {X 0,Y 216.121,Z 721.605,A -85,B 0,C 180,E1 -20768.541,E2 -20768.541} C_VEL
LIN {X 0,Y 217.982,Z 713.167,A -85,B 0,C 180,E1 -20771.192,E2 -20771.192} C_VEL
LIN {X 0,Y 219.889,Z 703.998,A -85,B 0,C 180,E1 -20773.502,E2 -20773.502} C_VEL
LIN {X 0,Y 221.871,Z 693.894,A -85,B 0,C 180,E1 -20775.549,E2 -20775.549} C_VEL
LIN {X 0,Y 223.727,Z 683.065,A -85,B 0,C 180,E1 -20777.298,E2 -20777.298} C_VEL
LIN {X 0,Y 225.583,Z 670.264,A -85,B 0,C 180,E1 -20778.886,E2 -20778.886} C_VEL
LIN {X 0,Y 226.911,Z 658.451,A -85,B 0,C 180,E1 -20779.988,E2 -20779.988} C_VEL
LIN {X 0,Y 227.966,Z 645.456,A -85,B 0,C 180,E1 -20780.835,E2 -20780.835} C_VEL
LIN {X 0,Y 228.834,Z 628.168,A -85,B 0,C 180,E1 -20781.501,E2 -20781.501} C_VEL
LIN {X 0,Y 230.931,Z 580.12,A -85,B 0,C 180,E1 -20783.094,E2 -20783.094} C_VEL
LIN {X 0,Y 221.315,Z 557.875,A -85,B 0,C 180,E1 -20785.162,E2 -20785.162} C_VEL
LIN {X 0,Y 214.352,Z 543.633,A -85,B 0,C 180,E1 -20786.711,E2 -20786.711} C_VEL
LIN {X 0,Y 214.218,Z 542.803,A -85,B 0,C 180,E1 -20786.826,E2 -20786.826} C_VEL
LIN {X 0,Y 214.548,Z 542.76,A -85,B 0,C 180,E1 -20790,E2 -20790} C_VEL
LIN {X 0,Y 214.444,Z 542.773,A -85,B 0,C 180,E1 -20791.878,E2 -20791.878} C_VEL
LIN {X 0,Y 214.246,Z 542.797,A -85,B 0,C 180,E1 -20797.54,E2 -20797.54} C_VEL
LIN {X 0,Y 214.045,Z 542.82,A -85,B 0,C 180,E1 -20801.362,E2 -20801.362} C_VEL
LIN {X 0,Y 213.931,Z 542.835,A -85,B 0,C 180,E1 -20805.237,E2 -20805.237} C_VEL
LIN {X 0,Y 213.837,Z 542.846,A -85,B 0,C 180,E1 -20809.187,E2 -20809.187} C_VEL
LIN {X 0,Y 213.844,Z 542.847,A -85,B 0,C 180,E1 -20813.227,E2 -20813.227} C_VEL
LIN {X 0,Y 213.825,Z 542.849,A -85,B 0,C 180,E1 -20817.45,E2 -20817.45} C_VEL
LIN {X 0,Y 213.776,Z 542.855,A -85,B 0,C 180,E1 -20821.735,E2 -20821.735} C_VEL
LIN {X 0,Y 213.75,Z 542.857,A -85,B 0,C 180,E1 -20826.286,E2 -20826.286} C_VEL
LIN {X 0,Y 213.82,Z 542.847,A -85,B 0,C 180,E1 -20831.099,E2 -20831.099} C_VEL
LIN {X 0,Y 213.832,Z 542.847,A -85,B 0,C 180,E1 -20833.693,E2 -20833.693} C_VEL
LIN {X 0,Y 213.836,Z 542.843,A -85,B 0,C 180,E1 -20836.356,E2 -20836.356} C_VEL
LIN {X 0,Y 213.779,Z 542.855,A -85,B 0,C 180,E1 -20841.346,E2 -20841.346} C_VEL
LIN {X 0,Y 213.764,Z 542.85,A -85,B 0,C 180,E1 -20846.02,E2 -20846.02} C_VEL
LIN {X 0,Y 213.776,Z 542.849,A -85,B 0,C 180,E1 -20850.454,E2 -20850.454} C_VEL
LIN {X 0,Y 213.793,Z 542.853,A -85,B 0,C 180,E1 -20854.702,E2 -20854.702} C_VEL
LIN {X 0,Y 213.797,Z 542.84,A -85,B 0,C 180,E1 -20858.803,E2 -20858.803} C_VEL
LIN {X 0,Y 213.938,Z 542.831,A -85,B 0,C 180,E1 -20862.804,E2 -20862.804} C_VEL
LIN {X 0,Y 213.948,Z 542.832,A -85,B 0,C 180,E1 -20866.707,E2 -20866.707} C_VEL
LIN {X 0,Y 214.162,Z 542.789,A -85,B 0,C 180,E1 -20870.557,E2 -20870.557} C_VEL
LIN {X 0,Y 214.223,Z 542.79,A -85,B 0,C 180,E1 -20872.46,E2 -20872.46} C_VEL
LIN {X 0,Y 214.442,Z 542.765,A -85,B 0,C 180,E1 -20878.123,E2 -20878.123} C_VEL
LIN {X 0,Y 214.55,Z 542.744,A -85,B 0,C 180,E1 -20880.001,E2 -20880.001} C_VEL
LIN {X 0,Y 214.477,Z 542.76,A -85,B 0,C 180,E1 -20881.879,E2 -20881.879} C_VEL
LIN {X 0,Y 214.205,Z 542.796,A -85,B 0,C 180,E1 -20887.542,E2 -20887.542} C_VEL
LIN {X 0,Y 213.995,Z 542.824,A -85,B 0,C 180,E1 -20891.365,E2 -20891.365} C_VEL
LIN {X 0,Y 213.93,Z 542.835,A -85,B 0,C 180,E1 -20895.238,E2 -20895.238} C_VEL
LIN {X 0,Y 213.837,Z 542.846,A -85,B 0,C 180,E1 -20899.189,E2 -20899.189} C_VEL
LIN {X 0,Y 213.845,Z 542.844,A -85,B 0,C 180,E1 -20903.228,E2 -20903.228} C_VEL
LIN {X 0,Y 213.827,Z 542.851,A -85,B 0,C 180,E1 -20907.451,E2 -20907.451} C_VEL
LIN {X 0,Y 213.778,Z 542.857,A -85,B 0,C 180,E1 -20911.737,E2 -20911.737} C_VEL
LIN {X 0,Y 213.747,Z 542.859,A -85,B 0,C 180,E1 -20916.289,E2 -20916.289} C_VEL
LIN {X 0,Y 213.725,Z 542.862,A -85,B 0,C 180,E1 -20921.123,E2 -20921.123} C_VEL
LIN {X 0,Y 213.72,Z 542.859,A -85,B 0,C 180,E1 -20924.356,E2 -20924.356} C_VEL
LIN {X 0,Y 213.826,Z 542.851,A -85,B 0,C 180,E1 -20928.746,E2 -20928.746} C_VEL
LIN {X 0,Y 214.286,Z 544.817,A -85,B 0,C 180,E1 -20929.657,E2 -20929.657} C_VEL
LIN {X 0,Y 214.129,Z 546.976,A -85,B 0,C 180,E1 -20930.545,E2 -20930.545} C_VEL
LIN {X 0,Y 212.032,Z 550.908,A -85,B 0,C 180,E1 -20931.904,E2 -20931.904} C_VEL
LIN {X 0,Y 209.918,Z 554.887,A -85,B 0,C 180,E1 -20933.288,E2 -20933.288} C_VEL
LIN {X 0,Y 209.775,Z 557.115,A -85,B 0,C 180,E1 -20934.197,E2 -20934.197} C_VEL
LIN {X 0,Y 210.431,Z 559.128,A -85,B 0,C 180,E1 -20934.449,E2 -20934.449} C_VEL
LIN {X 0,Y 217.884,Z 578.191,A -85,B 0,C 180,E1 -20936.28,E2 -20936.28} C_VEL
LIN {X 0,Y 219.421,Z 583.32,A -85,B 0,C 180,E1 -20936.689,E2 -20936.689} C_VEL
LIN {X 0,Y 223.328,Z 617.417,A -85,B 0,C 180,E1 -20938.531,E2 -20938.531} C_VEL
LIN {X 0,Y 221.091,Z 666.998,A -85,B 0,C 180,E1 -20940.285,E2 -20940.285} C_VEL
LIN {X 0,Y 219.844,Z 680.313,A -85,B 0,C 180,E1 -20941.085,E2 -20941.085} C_VEL
LIN {X 0,Y 218.217,Z 692.598,A -85,B 0,C 180,E1 -20942.161,E2 -20942.161} C_VEL
LIN {X 0,Y 216.364,Z 703.699,A -85,B 0,C 180,E1 -20943.473,E2 -20943.473} C_VEL
LIN {X 0,Y 214.142,Z 715.311,A -85,B 0,C 180,E1 -20945.264,E2 -20945.264} C_VEL
LIN {X 0,Y 211.907,Z 725.804,A -85,B 0,C 180,E1 -20947.323,E2 -20947.323} C_VEL
LIN {X 0,Y 209.89,Z 735.184,A -85,B 0,C 180,E1 -20949.648,E2 -20949.648} C_VEL
LIN {X 0,Y 208.062,Z 743.72,A -85,B 0,C 180,E1 -20952.302,E2 -20952.302} C_VEL
LIN {X 0,Y 206.509,Z 751.185,A -85,B 0,C 180,E1 -20955.212,E2 -20955.212} C_VEL
LIN {X 0,Y 205.406,Z 757.144,A -85,B 0,C 180,E1 -20958.154,E2 -20958.154} C_VEL
LIN {X 0,Y 204.848,Z 761.813,A -85,B 0,C 180,E1 -20961.119,E2 -20961.119} C_VEL
LIN {X 0,Y 204.718,Z 765.82,A -85,B 0,C 180,E1 -20964.617,E2 -20964.617} C_VEL
LIN {X 0,Y 204.726,Z 768.339,A -85,B 0,C 180,E1 -20968.033,E2 -20968.033} C_VEL
LIN {X 0,Y 204.777,Z 769.207,A -85,B 0,C 180,E1 -20970,E2 -20970} C_VEL
LIN {X 0,Y 204.689,Z 769.642,A -85,B 0,C 180,E1 -20971.968,E2 -20971.968} C_VEL
LIN {X 0,Y 204.493,Z 769.216,A -85,B 0,C 180,E1 -20975.918,E2 -20975.918} C_VEL
LIN {X 0,Y 204.909,Z 767.23,A -85,B 0,C 180,E1 -20979.874,E2 -20979.874} C_VEL
LIN {X 0,Y 205.745,Z 764.635,A -85,B 0,C 180,E1 -20982.828,E2 -20982.828} C_VEL
LIN {X 0,Y 207.179,Z 761.074,A -85,B 0,C 180,E1 -20985.746,E2 -20985.746} C_VEL
LIN {X 0,Y 209.126,Z 756.46,A -85,B 0,C 180,E1 -20988.618,E2 -20988.618} C_VEL
LIN {X 0,Y 211.666,Z 750.672,A -85,B 0,C 180,E1 -20991.422,E2 -20991.422} C_VEL
LIN {X 0,Y 214.552,Z 743.503,A -85,B 0,C 180,E1 -20994.17,E2 -20994.17} C_VEL
LIN {X 0,Y 218.119,Z 734.615,A -85,B 0,C 180,E1 -20996.813,E2 -20996.813} C_VEL
LIN {X 0,Y 221.858,Z 724.621,A -85,B 0,C 180,E1 -20999.146,E2 -20999.146} C_VEL
LIN {X 0,Y 225.58,Z 713.293,A -85,B 0,C 180,E1 -21001.194,E2 -21001.194} C_VEL
LIN {X 0,Y 228.888,Z 701.969,A -85,B 0,C 180,E1 -21002.763,E2 -21002.763} C_VEL
LIN {X 0,Y 231.714,Z 690.32,A -85,B 0,C 180,E1 -21004.001,E2 -21004.001} C_VEL
LIN {X 0,Y 234.335,Z 676.965,A -85,B 0,C 180,E1 -21005.001,E2 -21005.001} C_VEL
LIN {X 0,Y 236.077,Z 663.564,A -85,B 0,C 180,E1 -21005.703,E2 -21005.703} C_VEL
LIN {X 0,Y 238.906,Z 620.558,A -85,B 0,C 180,E1 -21007.152,E2 -21007.152} C_VEL
LIN {X 0,Y 237.542,Z 604.278,A -85,B 0,C 180,E1 -21008.304,E2 -21008.304} C_VEL
LIN {X 0,Y 236.93,Z 601.276,A -85,B 0,C 180,E1 -21008.618,E2 -21008.618} C_VEL
LIN {X 0,Y 232.357,Z 590.405,A -85,B 0,C 180,E1 -21010.456,E2 -21010.456} C_VEL
LIN {X 0,Y 227.597,Z 580.453,A -85,B 0,C 180,E1 -21012.502,E2 -21012.502} C_VEL
LIN {X 0,Y 223.99,Z 574.182,A -85,B 0,C 180,E1 -21014.111,E2 -21014.111} C_VEL
LIN {X 0,Y 221.249,Z 569.431,A -85,B 0,C 180,E1 -21015.456,E2 -21015.456} C_VEL
LIN {X 0,Y 217.819,Z 563.919,A -85,B 0,C 180,E1 -21017.244,E2 -21017.244} C_VEL
LIN {X 0,Y 214.357,Z 558.533,A -85,B 0,C 180,E1 -21019.257,E2 -21019.257} C_VEL
LIN {X 0,Y 210.381,Z 553.197,A -85,B 0,C 180,E1 -21021.828,E2 -21021.828} C_VEL
LIN {X 0,Y 209.121,Z 550.985,A -85,B 0,C 180,E1 -21022.775,E2 -21022.775} C_VEL
LIN {X 0,Y 207.821,Z 546.885,A -85,B 0,C 180,E1 -21027.242,E2 -21027.242} C_VEL
LIN {X 0,Y 206.763,Z 543.722,A -85,B 0,C 180,E1 -21031.937,E2 -21031.937} C_VEL
LIN {X 0,Y 206.783,Z 543.72,A -85,B 0,C 180,E1 -21036.583,E2 -21036.583} C_VEL
LIN {X 0,Y 206.873,Z 543.708,A -85,B 0,C 180,E1 -21042.196,E2 -21042.196} C_VEL
LIN {X 0,Y 206.91,Z 543.702,A -85,B 0,C 180,E1 -21046.244,E2 -21046.244} C_VEL
LIN {X 0,Y 207.102,Z 543.677,A -85,B 0,C 180,E1 -21050.23,E2 -21050.23} C_VEL
LIN {X 0,Y 207.173,Z 543.679,A -85,B 0,C 180,E1 -21052.2,E2 -21052.2} C_VEL
LIN {X 0,Y 207.42,Z 543.732,A -85,B 0,C 180,E1 -21058.3,E2 -21058.3} C_VEL
LIN {X 0,Y 208.119,Z 545.945,A -85,B 0,C 180,E1 -21059.032,E2 -21059.032} C_VEL
LIN {X 0,Y 210.41,Z 548.547,A -85,B 0,C 180,E1 -21060.716,E2 -21060.716} C_VEL
LIN {X 0,Y 211.829,Z 549.576,A -85,B 0,C 180,E1 -21061.606,E2 -21061.606} C_VEL
LIN {X 0,Y 213.399,Z 552.648,A -85,B 0,C 180,E1 -21062.713,E2 -21062.713} C_VEL
LIN {X 0,Y 215.983,Z 555.196,A -85,B 0,C 180,E1 -21064.198,E2 -21064.198} C_VEL
LIN {X 0,Y 218.345,Z 558.643,A -85,B 0,C 180,E1 -21065.54,E2 -21065.54} C_VEL
LIN {X 0,Y 219.811,Z 560.189,A -85,B 0,C 180,E1 -21066.266,E2 -21066.266} C_VEL
LIN {X 0,Y 223.449,Z 565.583,A -85,B 0,C 180,E1 -21068.065,E2 -21068.065} C_VEL
LIN {X 0,Y 226.549,Z 570.097,A -85,B 0,C 180,E1 -21069.463,E2 -21069.463} C_VEL
LIN {X 0,Y 231.492,Z 577.764,A -85,B 0,C 180,E1 -21071.52,E2 -21071.52} C_VEL
LIN {X 0,Y 237.24,Z 587.913,A -85,B 0,C 180,E1 -21073.708,E2 -21073.708} C_VEL
LIN {X 0,Y 240.476,Z 594.847,A -85,B 0,C 180,E1 -21074.909,E2 -21074.909} C_VEL
LIN {X 0,Y 236.929,Z 645.746,A -85,B 0,C 180,E1 -21076.603,E2 -21076.603} C_VEL
LIN {X 0,Y 235.319,Z 659.208,A -85,B 0,C 180,E1 -21077.376,E2 -21077.376} C_VEL
LIN {X 0,Y 233.319,Z 671.593,A -85,B 0,C 180,E1 -21078.437,E2 -21078.437} C_VEL
LIN {X 0,Y 230.785,Z 683.241,A -85,B 0,C 180,E1 -21079.775,E2 -21079.775} C_VEL
LIN {X 0,Y 227.562,Z 694.976,A -85,B 0,C 180,E1 -21081.51,E2 -21081.51} C_VEL
LIN {X 0,Y 224.206,Z 705.463,A -85,B 0,C 180,E1 -21083.53,E2 -21083.53} C_VEL
LIN {X 0,Y 220.682,Z 715.04,A -85,B 0,C 180,E1 -21085.888,E2 -21085.888} C_VEL
LIN {X 0,Y 217.469,Z 722.784,A -85,B 0,C 180,E1 -21088.282,E2 -21088.282} C_VEL
LIN {X 0,Y 214.548,Z 729.258,A -85,B 0,C 180,E1 -21090.796,E2 -21090.796} C_VEL
LIN {X 0,Y 211.63,Z 735.361,A -85,B 0,C 180,E1 -21093.881,E2 -21093.881} C_VEL
LIN {X 0,Y 209.094,Z 740.25,A -85,B 0,C 180,E1 -21097.228,E2 -21097.228} C_VEL
LIN {X 0,Y 207.459,Z 743.202,A -85,B 0,C 180,E1 -21100.064,E2 -21100.064} C_VEL
LIN {X 0,Y 206.171,Z 745.251,A -85,B 0,C 180,E1 -21102.98,E2 -21102.98} C_VEL
LIN {X 0,Y 205.047,Z 746.549,A -85,B 0,C 180,E1 -21106.726,E2 -21106.726} C_VEL
LIN {X 0,Y 204.591,Z 746.586,A -85,B 0,C 180,E1 -21109.258,E2 -21109.258} C_VEL
LIN {X 0,Y 204.373,Z 745.786,A -85,B 0,C 180,E1 -21112.27,E2 -21112.27} C_VEL
LIN {X 0,Y 204.528,Z 743.827,A -85,B 0,C 180,E1 -21115.555,E2 -21115.555} C_VEL
LIN {X 0,Y 205.172,Z 740.405,A -85,B 0,C 180,E1 -21119.083,E2 -21119.083} C_VEL
LIN {X 0,Y 206.116,Z 735.746,A -85,B 0,C 180,E1 -21122.438,E2 -21122.438} C_VEL
LIN {X 0,Y 207.312,Z 730.15,A -85,B 0,C 180,E1 -21125.464,E2 -21125.464} C_VEL
LIN {X 0,Y 209.031,Z 722.499,A -85,B 0,C 180,E1 -21128.679,E2 -21128.679} C_VEL
LIN {X 0,Y 210.605,Z 715.545,A -85,B 0,C 180,E1 -21131.013,E2 -21131.013} C_VEL
LIN {X 0,Y 212.606,Z 706.608,A -85,B 0,C 180,E1 -21133.46,E2 -21133.46} C_VEL
LIN {X 0,Y 214.75,Z 695.861,A -85,B 0,C 180,E1 -21135.792,E2 -21135.792} C_VEL
LIN {X 0,Y 216.818,Z 684.826,A -85,B 0,C 180,E1 -21137.68,E2 -21137.68} C_VEL
LIN {X 0,Y 218.571,Z 673.277,A -85,B 0,C 180,E1 -21139.229,E2 -21139.229} C_VEL
LIN {X 0,Y 220.1,Z 661.001,A -85,B 0,C 180,E1 -21140.466,E2 -21140.466} C_VEL
LIN {X 0,Y 221.256,Z 647.82,A -85,B 0,C 180,E1 -21141.42,E2 -21141.42} C_VEL
LIN {X 0,Y 222.112,Z 633.114,A -85,B 0,C 180,E1 -21142.054,E2 -21142.054} C_VEL
LIN {X 0,Y 224.511,Z 582.082,A -85,B 0,C 180,E1 -21143.784,E2 -21143.784} C_VEL
LIN {X 0,Y 215.438,Z 560.981,A -85,B 0,C 180,E1 -21145.822,E2 -21145.822} C_VEL
LIN {X 0,Y 207.562,Z 544.909,A -85,B 0,C 180,E1 -21147.65,E2 -21147.65} C_VEL
LIN {X 0,Y 207.317,Z 543.661,A -85,B 0,C 180,E1 -21147.784,E2 -21147.784} C_VEL
LIN {X 0,Y 207.513,Z 543.637,A -85,B 0,C 180,E1 -21150,E2 -21150} C_VEL
LIN {X 0,Y 207.381,Z 543.653,A -85,B 0,C 180,E1 -21151.942,E2 -21151.942} C_VEL
LIN {X 0,Y 207.186,Z 543.676,A -85,B 0,C 180,E1 -21157.798,E2 -21157.798} C_VEL
LIN {X 0,Y 206.981,Z 543.699,A -85,B 0,C 180,E1 -21161.755,E2 -21161.755} C_VEL
LIN {X 0,Y 206.864,Z 543.714,A -85,B 0,C 180,E1 -21165.771,E2 -21165.771} C_VEL
LIN {X 0,Y 206.781,Z 543.723,A -85,B 0,C 180,E1 -21169.869,E2 -21169.869} C_VEL
LIN {X 0,Y 206.76,Z 543.727,A -85,B 0,C 180,E1 -21174.072,E2 -21174.072} C_VEL
LIN {X 0,Y 206.741,Z 543.731,A -85,B 0,C 180,E1 -21178.419,E2 -21178.419} C_VEL
LIN {X 0,Y 206.705,Z 543.736,A -85,B 0,C 180,E1 -21182.956,E2 -21182.956} C_VEL
LIN {X 0,Y 206.722,Z 543.728,A -85,B 0,C 180,E1 -21187.73,E2 -21187.73} C_VEL
LIN {X 0,Y 206.745,Z 543.73,A -85,B 0,C 180,E1 -21191.597,E2 -21191.597} C_VEL
LIN {X 0,Y 206.742,Z 543.727,A -85,B 0,C 180,E1 -21195.55,E2 -21195.55} C_VEL
LIN {X 0,Y 206.724,Z 543.728,A -85,B 0,C 180,E1 -21199.765,E2 -21199.765} C_VEL
LIN {X 0,Y 206.721,Z 543.732,A -85,B 0,C 180,E1 -21202.27,E2 -21202.27} C_VEL
LIN {X 0,Y 206.704,Z 543.724,A -85,B 0,C 180,E1 -21207.045,E2 -21207.045} C_VEL
LIN {X 0,Y 206.762,Z 543.727,A -85,B 0,C 180,E1 -21212.097,E2 -21212.097} C_VEL
LIN {X 0,Y 206.749,Z 543.727,A -85,B 0,C 180,E1 -21216.605,E2 -21216.605} C_VEL
LIN {X 0,Y 206.867,Z 543.71,A -85,B 0,C 180,E1 -21222.197,E2 -21222.197} C_VEL
LIN {X 0,Y 206.89,Z 543.71,A -85,B 0,C 180,E1 -21226.245,E2 -21226.245} C_VEL
LIN {X 0,Y 207.101,Z 543.667,A -85,B 0,C 180,E1 -21230.232,E2 -21230.232} C_VEL
LIN {X 0,Y 207.163,Z 543.669,A -85,B 0,C 180,E1 -21232.202,E2 -21232.202} C_VEL
LIN {X 0,Y 207.378,Z 543.644,A -85,B 0,C 180,E1 -21238.059,E2 -21238.059} C_VEL
LIN {X 0,Y 207.514,Z 543.62,A -85,B 0,C 180,E1 -21240.001,E2 -21240.001} C_VEL
LIN {X 0,Y 207.41,Z 543.64,A -85,B 0,C 180,E1 -21241.943,E2 -21241.943} C_VEL
LIN {X 0,Y 207.145,Z 543.674,A -85,B 0,C 180,E1 -21247.801,E2 -21247.801} C_VEL
LIN {X 0,Y 206.921,Z 543.707,A -85,B 0,C 180,E1 -21251.76,E2 -21251.76} C_VEL
LIN {X 0,Y 206.863,Z 543.712,A -85,B 0,C 180,E1 -21255.772,E2 -21255.772} C_VEL
LIN {X 0,Y 206.781,Z 543.726,A -85,B 0,C 180,E1 -21259.87,E2 -21259.87} C_VEL
LIN {X 0,Y 206.761,Z 543.723,A -85,B 0,C 180,E1 -21264.073,E2 -21264.073} C_VEL
LIN {X 0,Y 206.743,Z 543.731,A -85,B 0,C 180,E1 -21268.42,E2 -21268.42} C_VEL
LIN {X 0,Y 206.708,Z 543.738,A -85,B 0,C 180,E1 -21272.957,E2 -21272.957} C_VEL
LIN {X 0,Y 206.721,Z 543.735,A -85,B 0,C 180,E1 -21275.322,E2 -21275.322} C_VEL
LIN {X 0,Y 206.669,Z 543.739,A -85,B 0,C 180,E1 -21280.251,E2 -21280.251} C_VEL
LIN {X 0,Y 206.709,Z 543.738,A -85,B 0,C 180,E1 -21285.562,E2 -21285.562} C_VEL
LIN {X 0,Y 206.788,Z 543.781,A -85,B 0,C 180,E1 -21288.048,E2 -21288.048} C_VEL
LIN {X 0,Y 209.122,Z 553.913,A -85,B 0,C 180,E1 -21292.777,E2 -21292.777} C_VEL
LIN {X 0,Y 209.775,Z 557.115,A -85,B 0,C 180,E1 -21294.197,E2 -21294.197} C_VEL
LIN {X 0,Y 212.054,Z 560.469,A -85,B 0,C 180,E1 -21294.731,E2 -21294.731} C_VEL
LIN {X 0,Y 213.68,Z 564.815,A -85,B 0,C 180,E1 -21295.131,E2 -21295.131} C_VEL
LIN {X 0,Y 214.394,Z 571.167,A -85,B 0,C 180,E1 -21295.501,E2 -21295.501} C_VEL
LIN {X 0,Y 214.392,Z 574.947,A -85,B 0,C 180,E1 -21295.587,E2 -21295.587} C_VEL
LIN {X 0,Y 213.401,Z 585.667,A -85,B 0,C 180,E1 -21295.992,E2 -21295.992} C_VEL
LIN {X 0,Y 213.49,Z 587.795,A -85,B 0,C 180,E1 -21296.104,E2 -21296.104} C_VEL
LIN {X 0,Y 216.839,Z 618.563,A -85,B 0,C 180,E1 -21297.81,E2 -21297.81} C_VEL
LIN {X 0,Y 214.533,Z 666.566,A -85,B 0,C 180,E1 -21299.553,E2 -21299.553} C_VEL
LIN {X 0,Y 213.288,Z 679.904,A -85,B 0,C 180,E1 -21300.38,E2 -21300.38} C_VEL
LIN {X 0,Y 211.596,Z 692.18,A -85,B 0,C 180,E1 -21301.481,E2 -21301.481} C_VEL
LIN {X 0,Y 209.692,Z 703.287,A -85,B 0,C 180,E1 -21302.829,E2 -21302.829} C_VEL
LIN {X 0,Y 207.389,Z 714.9,A -85,B 0,C 180,E1 -21304.67,E2 -21304.67} C_VEL
LIN {X 0,Y 205.085,Z 725.396,A -85,B 0,C 180,E1 -21306.791,E2 -21306.791} C_VEL
LIN {X 0,Y 203.036,Z 734.69,A -85,B 0,C 180,E1 -21309.165,E2 -21309.165} C_VEL
LIN {X 0,Y 201.629,Z 741.203,A -85,B 0,C 180,E1 -21311.191,E2 -21311.191} C_VEL
LIN {X 0,Y 199.894,Z 749.083,A -85,B 0,C 180,E1 -21314.189,E2 -21314.189} C_VEL
LIN {X 0,Y 198.738,Z 754.431,A -85,B 0,C 180,E1 -21316.711,E2 -21316.711} C_VEL
LIN {X 0,Y 197.959,Z 759.602,A -85,B 0,C 180,E1 -21319.775,E2 -21319.775} C_VEL
LIN {X 0,Y 197.595,Z 763.575,A -85,B 0,C 180,E1 -21322.849,E2 -21322.849} C_VEL
LIN {X 0,Y 197.606,Z 766.462,A -85,B 0,C 180,E1 -21325.921,E2 -21325.921} C_VEL
LIN {X 0,Y 197.658,Z 767.79,A -85,B 0,C 180,E1 -21327.962,E2 -21327.962} C_VEL
LIN {X 0,Y 197.707,Z 768.697,A -85,B 0,C 180,E1 -21330,E2 -21330} C_VEL
LIN {X 0,Y 197.614,Z 769.183,A -85,B 0,C 180,E1 -21332.038,E2 -21332.038} C_VEL
LIN {X 0,Y 197.407,Z 769.165,A -85,B 0,C 180,E1 -21334.543,E2 -21334.543} C_VEL
LIN {X 0,Y 197.562,Z 768.1,A -85,B 0,C 180,E1 -21338.18,E2 -21338.18} C_VEL
LIN {X 0,Y 197.893,Z 766.958,A -85,B 0,C 180,E1 -21340.228,E2 -21340.228} C_VEL
LIN {X 0,Y 198.789,Z 764.452,A -85,B 0,C 180,E1 -21343.285,E2 -21343.285} C_VEL
LIN {X 0,Y 200.326,Z 760.983,A -85,B 0,C 180,E1 -21346.299,E2 -21346.299} C_VEL
LIN {X 0,Y 202.383,Z 756.464,A -85,B 0,C 180,E1 -21349.262,E2 -21349.262} C_VEL
LIN {X 0,Y 205.021,Z 750.779,A -85,B 0,C 180,E1 -21352.152,E2 -21352.152} C_VEL
LIN {X 0,Y 208.09,Z 743.778,A -85,B 0,C 180,E1 -21354.971,E2 -21354.971} C_VEL
LIN {X 0,Y 211.842,Z 735.112,A -85,B 0,C 180,E1 -21357.675,E2 -21357.675} C_VEL
LIN {X 0,Y 215.345,Z 726.3,A -85,B 0,C 180,E1 -21359.847,E2 -21359.847} C_VEL
LIN {X 0,Y 219.184,Z 715.548,A -85,B 0,C 180,E1 -21361.941,E2 -21361.941} C_VEL
LIN {X 0,Y 222.634,Z 704.876,A -85,B 0,C 180,E1 -21363.533,E2 -21363.533} C_VEL
LIN {X 0,Y 225.718,Z 693.105,A -85,B 0,C 180,E1 -21364.898,E2 -21364.898} C_VEL
LIN {X 0,Y 228.59,Z 680,A -85,B 0,C 180,E1 -21365.993,E2 -21365.993} C_VEL
LIN {X 0,Y 230.611,Z 666.945,A -85,B 0,C 180,E1 -21366.754,E2 -21366.754} C_VEL
LIN {X 0,Y 232.102,Z 648.479,A -85,B 0,C 180,E1 -21367.456,E2 -21367.456} C_VEL
LIN {X 0,Y 233.917,Z 621.642,A -85,B 0,C 180,E1 -21368.364,E2 -21368.364} C_VEL
LIN {X 0,Y 232.74,Z 606.201,A -85,B 0,C 180,E1 -21369.494,E2 -21369.494} C_VEL
LIN {X 0,Y 231.676,Z 603.006,A -85,B 0,C 180,E1 -21369.965,E2 -21369.965} C_VEL
LIN {X 0,Y 227.67,Z 593.3,A -85,B 0,C 180,E1 -21371.715,E2 -21371.715} C_VEL
LIN {X 0,Y 223.437,Z 584.505,A -85,B 0,C 180,E1 -21373.659,E2 -21373.659} C_VEL
LIN {X 0,Y 219.933,Z 578.07,A -85,B 0,C 180,E1 -21375.387,E2 -21375.387} C_VEL
LIN {X 0,Y 217.861,Z 574.524,A -85,B 0,C 180,E1 -21376.466,E2 -21376.466} C_VEL
LIN {X 0,Y 215.04,Z 569.754,A -85,B 0,C 180,E1 -21378.039,E2 -21378.039} C_VEL
LIN {X 0,Y 211.229,Z 563.727,A -85,B 0,C 180,E1 -21380.413,E2 -21380.413} C_VEL
LIN {X 0,Y 208.046,Z 559.255,A -85,B 0,C 180,E1 -21382.615,E2 -21382.615} C_VEL
LIN {X 0,Y 206.559,Z 556.859,A -85,B 0,C 180,E1 -21383.8,E2 -21383.8} C_VEL
LIN {X 0,Y 202.201,Z 550.981,A -85,B 0,C 180,E1 -21387.85,E2 -21387.85} C_VEL
LIN {X 0,Y 201.269,Z 549.413,A -85,B 0,C 180,E1 -21388.998,E2 -21388.998} C_VEL
LIN {X 0,Y 200.455,Z 547.043,A -85,B 0,C 180,E1 -21392.884,E2 -21392.884} C_VEL
LIN {X 0,Y 199.709,Z 544.619,A -85,B 0,C 180,E1 -21398.585,E2 -21398.585} C_VEL
LIN {X 0,Y 199.835,Z 544.588,A -85,B 0,C 180,E1 -21401.721,E2 -21401.721} C_VEL
LIN {X 0,Y 199.844,Z 544.584,A -85,B 0,C 180,E1 -21405.748,E2 -21405.748} C_VEL
LIN {X 0,Y 200.065,Z 544.556,A -85,B 0,C 180,E1 -21410.904,E2 -21410.904} C_VEL
LIN {X 0,Y 200.139,Z 544.72,A -85,B 0,C 180,E1 -21411.988,E2 -21411.988} C_VEL
LIN {X 0,Y 200.947,Z 547.229,A -85,B 0,C 180,E1 -21413.346,E2 -21413.346} C_VEL
LIN {X 0,Y 202.926,Z 549.461,A -85,B 0,C 180,E1 -21415.53,E2 -21415.53} C_VEL
LIN {X 0,Y 205.403,Z 550.624,A -85,B 0,C 180,E1 -21417.634,E2 -21417.634} C_VEL
LIN {X 0,Y 206.909,Z 553.515,A -85,B 0,C 180,E1 -21419.026,E2 -21419.026} C_VEL
LIN {X 0,Y 209.601,Z 556.183,A -85,B 0,C 180,E1 -21420.96,E2 -21420.96} C_VEL
LIN {X 0,Y 211.617,Z 559.524,A -85,B 0,C 180,E1 -21422.378,E2 -21422.378} C_VEL
LIN {X 0,Y 213.656,Z 561.669,A -85,B 0,C 180,E1 -21423.594,E2 -21423.594} C_VEL
LIN {X 0,Y 216.173,Z 565.166,A -85,B 0,C 180,E1 -21425.063,E2 -21425.063} C_VEL
LIN {X 0,Y 217.429,Z 566.827,A -85,B 0,C 180,E1 -21425.744,E2 -21425.744} C_VEL
LIN {X 0,Y 220.616,Z 571.568,A -85,B 0,C 180,E1 -21427.377,E2 -21427.377} C_VEL
LIN {X 0,Y 224.976,Z 578.092,A -85,B 0,C 180,E1 -21429.42,E2 -21429.42} C_VEL
LIN {X 0,Y 229.263,Z 585.314,A -85,B 0,C 180,E1 -21431.26,E2 -21431.26} C_VEL
LIN {X 0,Y 233.638,Z 593.506,A -85,B 0,C 180,E1 -21433.018,E2 -21433.018} C_VEL
LIN {X 0,Y 235.463,Z 597.291,A -85,B 0,C 180,E1 -21433.72,E2 -21433.72} C_VEL
LIN {X 0,Y 231.93,Z 645.924,A -85,B 0,C 180,E1 -21435.371,E2 -21435.371} C_VEL
LIN {X 0,Y 230.182,Z 659.902,A -85,B 0,C 180,E1 -21436.19,E2 -21436.19} C_VEL
LIN {X 0,Y 228.11,Z 671.952,A -85,B 0,C 180,E1 -21437.239,E2 -21437.239} C_VEL
LIN {X 0,Y 225.466,Z 683.517,A -85,B 0,C 180,E1 -21438.585,E2 -21438.585} C_VEL
LIN {X 0,Y 222.065,Z 695.437,A -85,B 0,C 180,E1 -21440.372,E2 -21440.372} C_VEL
LIN {X 0,Y 218.57,Z 705.8,A -85,B 0,C 180,E1 -21442.392,E2 -21442.392} C_VEL
LIN {X 0,Y 214.798,Z 715.491,A -85,B 0,C 180,E1 -21444.814,E2 -21444.814} C_VEL
LIN {X 0,Y 211.342,Z 723.407,A -85,B 0,C 180,E1 -21447.326,E2 -21447.326} C_VEL
LIN {X 0,Y 208.235,Z 729.819,A -85,B 0,C 180,E1 -21449.894,E2 -21449.894} C_VEL
LIN {X 0,Y 204.951,Z 736.212,A -85,B 0,C 180,E1 -21453.274,E2 -21453.274} C_VEL
LIN {X 0,Y 202.162,Z 741.23,A -85,B 0,C 180,E1 -21456.912,E2 -21456.912} C_VEL
LIN {X 0,Y 200.582,Z 743.798,A -85,B 0,C 180,E1 -21459.573,E2 -21459.573} C_VEL
LIN {X 0,Y 199.34,Z 745.606,A -85,B 0,C 180,E1 -21462.237,E2 -21462.237} C_VEL
LIN {X 0,Y 198.369,Z 746.758,A -85,B 0,C 180,E1 -21465.118,E2 -21465.118} C_VEL
LIN {X 0,Y 197.635,Z 747.083,A -85,B 0,C 180,E1 -21468.31,E2 -21468.31} C_VEL
LIN {X 0,Y 197.307,Z 746.396,A -85,B 0,C 180,E1 -21471.592,E2 -21471.592} C_VEL
LIN {X 0,Y 197.398,Z 744.367,A -85,B 0,C 180,E1 -21475.275,E2 -21475.275} C_VEL
LIN {X 0,Y 197.942,Z 741.53,A -85,B 0,C 180,E1 -21478.442,E2 -21478.442} C_VEL
LIN {X 0,Y 198.885,Z 736.917,A -85,B 0,C 180,E1 -21482.056,E2 -21482.056} C_VEL
LIN {X 0,Y 199.997,Z 731.809,A -85,B 0,C 180,E1 -21485.06,E2 -21485.06} C_VEL
LIN {X 0,Y 201.435,Z 725.548,A -85,B 0,C 180,E1 -21487.973,E2 -21487.973} C_VEL
LIN {X 0,Y 203.257,Z 717.826,A -85,B 0,C 180,E1 -21490.824,E2 -21490.824} C_VEL
LIN {X 0,Y 205.314,Z 709.017,A -85,B 0,C 180,E1 -21493.423,E2 -21493.423} C_VEL
LIN {X 0,Y 207.45,Z 699.07,A -85,B 0,C 180,E1 -21495.782,E2 -21495.782} C_VEL
LIN {X 0,Y 209.598,Z 688.088,A -85,B 0,C 180,E1 -21497.836,E2 -21497.836} C_VEL
LIN {X 0,Y 211.459,Z 676.995,A -85,B 0,C 180,E1 -21499.468,E2 -21499.468} C_VEL
LIN {X 0,Y 213.153,Z 664.587,A -85,B 0,C 180,E1 -21500.872,E2 -21500.872} C_VEL
LIN {X 0,Y 214.411,Z 651.896,A -85,B 0,C 180,E1 -21501.907,E2 -21501.907} C_VEL
LIN {X 0,Y 215.34,Z 638.428,A -85,B 0,C 180,E1 -21502.614,E2 -21502.614} C_VEL
LIN {X 0,Y 218,Z 584.439,A -85,B 0,C 180,E1 -21504.502,E2 -21504.502} C_VEL
LIN {X 0,Y 217.088,Z 581.496,A -85,B 0,C 180,E1 -21504.742,E2 -21504.742} C_VEL
LIN {X 0,Y 209.189,Z 563.348,A -85,B 0,C 180,E1 -21506.602,E2 -21506.602} C_VEL
LIN {X 0,Y 200.566,Z 545.578,A -85,B 0,C 180,E1 -21508.714,E2 -21508.714} C_VEL
LIN {X 0,Y 200.368,Z 544.527,A -85,B 0,C 180,E1 -21508.87,E2 -21508.87} C_VEL
LIN {X 0,Y 200.32,Z 544.533,A -85,B 0,C 180,E1 -21512.011,E2 -21512.011} C_VEL
LIN {X 0,Y 200.13,Z 544.555,A -85,B 0,C 180,E1 -21518.075,E2 -21518.075} C_VEL
LIN {X 0,Y 199.912,Z 544.58,A -85,B 0,C 180,E1 -21522.177,E2 -21522.177} C_VEL
LIN {X 0,Y 199.802,Z 544.594,A -85,B 0,C 180,E1 -21526.343,E2 -21526.343} C_VEL
LIN {X 0,Y 199.697,Z 544.607,A -85,B 0,C 180,E1 -21530.605,E2 -21530.605} C_VEL
LIN {X 0,Y 199.67,Z 544.613,A -85,B 0,C 180,E1 -21534.984,E2 -21534.984} C_VEL
LIN {X 0,Y 199.671,Z 544.611,A -85,B 0,C 180,E1 -21539.522,E2 -21539.522} C_VEL
LIN {X 0,Y 199.66,Z 544.613,A -85,B 0,C 180,E1 -21542.352,E2 -21542.352} C_VEL
LIN {X 0,Y 199.649,Z 544.614,A -85,B 0,C 180,E1 -21546.756,E2 -21546.756} C_VEL
LIN {X 0,Y 199.698,Z 544.6,A -85,B 0,C 180,E1 -21549.306,E2 -21549.306} C_VEL
LIN {X 0,Y 199.696,Z 544.608,A -85,B 0,C 180,E1 -21552.35,E2 -21552.35} C_VEL
LIN {X 0,Y 199.69,Z 544.607,A -85,B 0,C 180,E1 -21555.261,E2 -21555.261} C_VEL
LIN {X 0,Y 199.674,Z 544.596,A -85,B 0,C 180,E1 -21558.031,E2 -21558.031} C_VEL
LIN {X 0,Y 199.697,Z 544.605,A -85,B 0,C 180,E1 -21560.736,E2 -21560.736} C_VEL
LIN {X 0,Y 199.63,Z 544.61,A -85,B 0,C 180,E1 -21565.718,E2 -21565.718} C_VEL
LIN {X 0,Y 199.699,Z 544.591,A -85,B 0,C 180,E1 -21568.138,E2 -21568.138} C_VEL
LIN {X 0,Y 199.682,Z 544.611,A -85,B 0,C 180,E1 -21572.772,E2 -21572.772} C_VEL
LIN {X 0,Y 199.709,Z 544.598,A -85,B 0,C 180,E1 -21577.227,E2 -21577.227} C_VEL
LIN {X 0,Y 199.791,Z 544.592,A -85,B 0,C 180,E1 -21581.759,E2 -21581.759} C_VEL
LIN {X 0,Y 199.83,Z 544.59,A -85,B 0,C 180,E1 -21585.749,E2 -21585.749} C_VEL
LIN {X 0,Y 200.066,Z 544.543,A -85,B 0,C 180,E1 -21589.885,E2 -21589.885} C_VEL
LIN {X 0,Y 200.031,Z 544.563,A -85,B 0,C 180,E1 -21593.951,E2 -21593.951} C_VEL
LIN {X 0,Y 200.318,Z 544.524,A -85,B 0,C 180,E1 -21597.99,E2 -21597.99} C_VEL
LIN {X 0,Y 200.478,Z 544.495,A -85,B 0,C 180,E1 -21600.001,E2 -21600.001} C_VEL
LIN {X 0,Y 200.346,Z 544.519,A -85,B 0,C 180,E1 -21602.011,E2 -21602.011} C_VEL
LIN {X 0,Y 200.092,Z 544.552,A -85,B 0,C 180,E1 -21608.078,E2 -21608.078} C_VEL
LIN {X 0,Y 199.871,Z 544.585,A -85,B 0,C 180,E1 -21612.181,E2 -21612.181} C_VEL
LIN {X 0,Y 199.801,Z 544.591,A -85,B 0,C 180,E1 -21616.345,E2 -21616.345} C_VEL
LIN {X 0,Y 199.697,Z 544.609,A -85,B 0,C 180,E1 -21620.607,E2 -21620.607} C_VEL
LIN {X 0,Y 199.671,Z 544.607,A -85,B 0,C 180,E1 -21624.986,E2 -21624.986} C_VEL
LIN {X 0,Y 199.673,Z 544.609,A -85,B 0,C 180,E1 -21629.524,E2 -21629.524} C_VEL
LIN {X 0,Y 199.663,Z 544.614,A -85,B 0,C 180,E1 -21632.353,E2 -21632.353} C_VEL
LIN {X 0,Y 199.639,Z 544.617,A -85,B 0,C 180,E1 -21636.761,E2 -21636.761} C_VEL
LIN {X 0,Y 199.639,Z 544.618,A -85,B 0,C 180,E1 -21639.322,E2 -21639.322} C_VEL
LIN {X 0,Y 199.631,Z 544.618,A -85,B 0,C 180,E1 -21644.758,E2 -21644.758} C_VEL
LIN {X 0,Y 199.763,Z 544.705,A -85,B 0,C 180,E1 -21647.302,E2 -21647.302} C_VEL
LIN {X 0,Y 202.093,Z 554.878,A -85,B 0,C 180,E1 -21652.242,E2 -21652.242} C_VEL
LIN {X 0,Y 202.586,Z 557.17,A -85,B 0,C 180,E1 -21653.191,E2 -21653.191} C_VEL
LIN {X 0,Y 211.611,Z 580.231,A -85,B 0,C 180,E1 -21655.526,E2 -21655.526} C_VEL
LIN {X 0,Y 213.167,Z 585.241,A -85,B 0,C 180,E1 -21655.952,E2 -21655.952} C_VEL
LIN {X 0,Y 213.49,Z 587.795,A -85,B 0,C 180,E1 -21656.104,E2 -21656.104} C_VEL
LIN {X 0,Y 213.522,Z 595.552,A -85,B 0,C 180,E1 -21656.436,E2 -21656.436} C_VEL
LIN {X 0,Y 210.389,Z 619.013,A -85,B 0,C 180,E1 -21657.017,E2 -21657.017} C_VEL
LIN {X 0,Y 208.031,Z 666.147,A -85,B 0,C 180,E1 -21658.778,E2 -21658.778} C_VEL
LIN {X 0,Y 206.842,Z 678.75,A -85,B 0,C 180,E1 -21659.571,E2 -21659.571} C_VEL
LIN {X 0,Y 205.011,Z 691.764,A -85,B 0,C 180,E1 -21660.758,E2 -21660.758} C_VEL
LIN {X 0,Y 203.048,Z 702.876,A -85,B 0,C 180,E1 -21662.144,E2 -21662.144} C_VEL
LIN {X 0,Y 200.662,Z 714.488,A -85,B 0,C 180,E1 -21664.037,E2 -21664.037} C_VEL
LIN {X 0,Y 198.283,Z 724.988,A -85,B 0,C 180,E1 -21666.224,E2 -21666.224} C_VEL
LIN {X 0,Y 196.151,Z 734.314,A -85,B 0,C 180,E1 -21668.683,E2 -21668.683} C_VEL
LIN {X 0,Y 194.781,Z 740.199,A -85,B 0,C 180,E1 -21670.564,E2 -21670.564} C_VEL
LIN {X 0,Y 193.007,Z 748.1,A -85,B 0,C 180,E1 -21673.609,E2 -21673.609} C_VEL
LIN {X 0,Y 191.799,Z 753.527,A -85,B 0,C 180,E1 -21676.221,E2 -21676.221} C_VEL
LIN {X 0,Y 190.941,Z 758.822,A -85,B 0,C 180,E1 -21679.395,E2 -21679.395} C_VEL
LIN {X 0,Y 190.519,Z 762.889,A -85,B 0,C 180,E1 -21682.582,E2 -21682.582} C_VEL
LIN {X 0,Y 190.535,Z 765.857,A -85,B 0,C 180,E1 -21685.769,E2 -21685.769} C_VEL
LIN {X 0,Y 190.592,Z 767.241,A -85,B 0,C 180,E1 -21687.887,E2 -21687.887} C_VEL
LIN {X 0,Y 190.639,Z 768.185,A -85,B 0,C 180,E1 -21690,E2 -21690} C_VEL
LIN {X 0,Y 190.54,Z 768.708,A -85,B 0,C 180,E1 -21692.114,E2 -21692.114} C_VEL
LIN {X 0,Y 190.333,Z 768.804,A -85,B 0,C 180,E1 -21694.45,E2 -21694.45} C_VEL
LIN {X 0,Y 190.506,Z 767.789,A -85,B 0,C 180,E1 -21698.486,E2 -21698.486} C_VEL
LIN {X 0,Y 191.476,Z 765.201,A -85,B 0,C 180,E1 -21702.722,E2 -21702.722} C_VEL
LIN {X 0,Y 192.869,Z 762.142,A -85,B 0,C 180,E1 -21705.86,E2 -21705.86} C_VEL
LIN {X 0,Y 194.895,Z 758.086,A -85,B 0,C 180,E1 -21708.937,E2 -21708.937} C_VEL
LIN {X 0,Y 197.578,Z 752.938,A -85,B 0,C 180,E1 -21711.931,E2 -21711.931} C_VEL
LIN {X 0,Y 200.514,Z 746.552,A -85,B 0,C 180,E1 -21714.872,E2 -21714.872} C_VEL
LIN {X 0,Y 204.222,Z 738.638,A -85,B 0,C 180,E1 -21717.682,E2 -21717.682} C_VEL
LIN {X 0,Y 208.547,Z 728.838,A -85,B 0,C 180,E1 -21720.364,E2 -21720.364} C_VEL
LIN {X 0,Y 212.417,Z 718.81,A -85,B 0,C 180,E1 -21722.523,E2 -21722.523} C_VEL
LIN {X 0,Y 216.354,Z 707.597,A -85,B 0,C 180,E1 -21724.36,E2 -21724.36} C_VEL
LIN {X 0,Y 219.542,Z 696.773,A -85,B 0,C 180,E1 -21725.747,E2 -21725.747} C_VEL
LIN {X 0,Y 222.502,Z 684.949,A -85,B 0,C 180,E1 -21726.879,E2 -21726.879} C_VEL
LIN {X 0,Y 224.947,Z 672.234,A -85,B 0,C 180,E1 -21727.745,E2 -21727.745} C_VEL
LIN {X 0,Y 226.505,Z 658.507,A -85,B 0,C 180,E1 -21728.404,E2 -21728.404} C_VEL
LIN {X 0,Y 229.068,Z 622.658,A -85,B 0,C 180,E1 -21729.638,E2 -21729.638} C_VEL
LIN {X 0,Y 228.124,Z 608.59,A -85,B 0,C 180,E1 -21730.688,E2 -21730.688} C_VEL
LIN {X 0,Y 223.746,Z 597.654,A -85,B 0,C 180,E1 -21732.737,E2 -21732.737} C_VEL
LIN {X 0,Y 219.801,Z 589.237,A -85,B 0,C 180,E1 -21734.678,E2 -21734.678} C_VEL
LIN {X 0,Y 215.535,Z 581.067,A -85,B 0,C 180,E1 -21736.973,E2 -21736.973} C_VEL
LIN {X 0,Y 212.196,Z 575.37,A -85,B 0,C 180,E1 -21738.948,E2 -21738.948} C_VEL
LIN {X 0,Y 208.681,Z 569.688,A -85,B 0,C 180,E1 -21741.26,E2 -21741.26} C_VEL
LIN {X 0,Y 205.489,Z 564.704,A -85,B 0,C 180,E1 -21743.69,E2 -21743.69} C_VEL
LIN {X 0,Y 204.383,Z 563.074,A -85,B 0,C 180,E1 -21744.615,E2 -21744.615} C_VEL
LIN {X 0,Y 199.499,Z 555.952,A -85,B 0,C 180,E1 -21749.72,E2 -21749.72} C_VEL
LIN {X 0,Y 196.078,Z 551.721,A -85,B 0,C 180,E1 -21755.568,E2 -21755.568} C_VEL
LIN {X 0,Y 195.271,Z 550.142,A -85,B 0,C 180,E1 -21758.904,E2 -21758.904} C_VEL
LIN {X 0,Y 195.148,Z 549.944,A -85,B 0,C 180,E1 -21763.254,E2 -21763.254} C_VEL
LIN {X 0,Y 198.611,Z 551.599,A -85,B 0,C 180,E1 -21771.395,E2 -21771.395} C_VEL
LIN {X 0,Y 199.706,Z 554.363,A -85,B 0,C 180,E1 -21773.178,E2 -21773.178} C_VEL
LIN {X 0,Y 201.806,Z 556.519,A -85,B 0,C 180,E1 -21775.505,E2 -21775.505} C_VEL
LIN {X 0,Y 203.658,Z 557.592,A -85,B 0,C 180,E1 -21777.151,E2 -21777.151} C_VEL
LIN {X 0,Y 205.56,Z 560.686,A -85,B 0,C 180,E1 -21778.882,E2 -21778.882} C_VEL
LIN {X 0,Y 207.474,Z 562.671,A -85,B 0,C 180,E1 -21780.303,E2 -21780.303} C_VEL
LIN {X 0,Y 209.66,Z 566.185,A -85,B 0,C 180,E1 -21781.92,E2 -21781.92} C_VEL
LIN {X 0,Y 211.321,Z 568.012,A -85,B 0,C 180,E1 -21782.949,E2 -21782.949} C_VEL
LIN {X 0,Y 214.05,Z 571.702,A -85,B 0,C 180,E1 -21784.589,E2 -21784.589} C_VEL
LIN {X 0,Y 217.761,Z 577.452,A -85,B 0,C 180,E1 -21786.644,E2 -21786.644} C_VEL
LIN {X 0,Y 222.281,Z 584.554,A -85,B 0,C 180,E1 -21788.88,E2 -21788.88} C_VEL
LIN {X 0,Y 226.549,Z 591.963,A -85,B 0,C 180,E1 -21790.786,E2 -21790.786} C_VEL
LIN {X 0,Y 230.464,Z 599.785,A -85,B 0,C 180,E1 -21792.457,E2 -21792.457} C_VEL
LIN {X 0,Y 228.93,Z 621.538,A -85,B 0,C 180,E1 -21793.21,E2 -21793.21} C_VEL
LIN {X 0,Y 226.977,Z 647.197,A -85,B 0,C 180,E1 -21794.138,E2 -21794.138} C_VEL
LIN {X 0,Y 225.143,Z 660.917,A -85,B 0,C 180,E1 -21794.961,E2 -21794.961} C_VEL
LIN {X 0,Y 222.861,Z 673.24,A -85,B 0,C 180,E1 -21796.066,E2 -21796.066} C_VEL
LIN {X 0,Y 220.162,Z 684.419,A -85,B 0,C 180,E1 -21797.401,E2 -21797.401} C_VEL
LIN {X 0,Y 216.789,Z 695.568,A -85,B 0,C 180,E1 -21799.099,E2 -21799.099} C_VEL
LIN {X 0,Y 213.376,Z 705.262,A -85,B 0,C 180,E1 -21800.987,E2 -21800.987} C_VEL
LIN {X 0,Y 210.196,Z 713.199,A -85,B 0,C 180,E1 -21802.913,E2 -21802.913} C_VEL
LIN {X 0,Y 206.437,Z 721.603,A -85,B 0,C 180,E1 -21805.451,E2 -21805.451} C_VEL
LIN {X 0,Y 203.049,Z 728.397,A -85,B 0,C 180,E1 -21808.045,E2 -21808.045} C_VEL
LIN {X 0,Y 199.521,Z 735,A -85,B 0,C 180,E1 -21811.332,E2 -21811.332} C_VEL
LIN {X 0,Y 196.388,Z 740.312,A -85,B 0,C 180,E1 -21814.929,E2 -21814.929} C_VEL
LIN {X 0,Y 194.395,Z 743.476,A -85,B 0,C 180,E1 -21817.922,E2 -21817.922} C_VEL
LIN {X 0,Y 192.746,Z 745.739,A -85,B 0,C 180,E1 -21821.019,E2 -21821.019} C_VEL
LIN {X 0,Y 191.543,Z 747.084,A -85,B 0,C 180,E1 -21824.196,E2 -21824.196} C_VEL
LIN {X 0,Y 190.522,Z 747.452,A -85,B 0,C 180,E1 -21828.397,E2 -21828.397} C_VEL
LIN {X 0,Y 190.235,Z 746.887,A -85,B 0,C 180,E1 -21831.095,E2 -21831.095} C_VEL
LIN {X 0,Y 190.221,Z 745.298,A -85,B 0,C 180,E1 -21834.371,E2 -21834.371} C_VEL
LIN {X 0,Y 190.733,Z 742.434,A -85,B 0,C 180,E1 -21837.937,E2 -21837.937} C_VEL
LIN {X 0,Y 191.65,Z 738.035,A -85,B 0,C 180,E1 -21841.653,E2 -21841.653} C_VEL
LIN {X 0,Y 192.747,Z 732.985,A -85,B 0,C 180,E1 -21844.844,E2 -21844.844} C_VEL
LIN {X 0,Y 194.431,Z 726.032,A -85,B 0,C 180,E1 -21848.254,E2 -21848.254} C_VEL
LIN {X 0,Y 196.292,Z 718.344,A -85,B 0,C 180,E1 -21851.202,E2 -21851.202} C_VEL
LIN {X 0,Y 198.592,Z 708.849,A -85,B 0,C 180,E1 -21854.082,E2 -21854.082} C_VEL
LIN {X 0,Y 200.534,Z 700.159,A -85,B 0,C 180,E1 -21856.206,E2 -21856.206} C_VEL
LIN {X 0,Y 202.644,Z 689.87,A -85,B 0,C 180,E1 -21858.244,E2 -21858.244} C_VEL
LIN {X 0,Y 204.791,Z 677.679,A -85,B 0,C 180,E1 -21860.12,E2 -21860.12} C_VEL
LIN {X 0,Y 206.539,Z 665.368,A -85,B 0,C 180,E1 -21861.563,E2 -21861.563} C_VEL
LIN {X 0,Y 207.867,Z 652.567,A -85,B 0,C 180,E1 -21862.65,E2 -21862.65} C_VEL
LIN {X 0,Y 208.837,Z 639.456,A -85,B 0,C 180,E1 -21863.367,E2 -21863.367} C_VEL
LIN {X 0,Y 211.541,Z 585.411,A -85,B 0,C 180,E1 -21865.322,E2 -21865.322} C_VEL
LIN {X 0,Y 203.716,Z 567.239,A -85,B 0,C 180,E1 -21867.23,E2 -21867.23} C_VEL
LIN {X 0,Y 194.148,Z 547.765,A -85,B 0,C 180,E1 -21869.673,E2 -21869.673} C_VEL
LIN {X 0,Y 193.44,Z 545.39,A -85,B 0,C 180,E1 -21869.935,E2 -21869.935} C_VEL
LIN {X 0,Y 192.978,Z 545.447,A -85,B 0,C 180,E1 -21874.177,E2 -21874.177} C_VEL
LIN {X 0,Y 193.077,Z 545.434,A -85,B 0,C 180,E1 -21878.372,E2 -21878.372} C_VEL
LIN {X 0,Y 192.851,Z 545.461,A -85,B 0,C 180,E1 -21882.63,E2 -21882.63} C_VEL
LIN {X 0,Y 192.755,Z 545.472,A -85,B 0,C 180,E1 -21886.959,E2 -21886.959} C_VEL
LIN {X 0,Y 192.634,Z 545.487,A -85,B 0,C 180,E1 -21891.397,E2 -21891.397} C_VEL
LIN {X 0,Y 192.661,Z 545.484,A -85,B 0,C 180,E1 -21894.225,E2 -21894.225} C_VEL
LIN {X 0,Y 192.646,Z 545.487,A -85,B 0,C 180,E1 -21898.892,E2 -21898.892} C_VEL
LIN {X 0,Y 192.597,Z 545.493,A -85,B 0,C 180,E1 -21903.185,E2 -21903.185} C_VEL
LIN {X 0,Y 192.609,Z 545.484,A -85,B 0,C 180,E1 -21908.337,E2 -21908.337} C_VEL
LIN {X 0,Y 192.629,Z 545.491,A -85,B 0,C 180,E1 -21913.141,E2 -21913.141} C_VEL
LIN {X 0,Y 192.616,Z 545.48,A -85,B 0,C 180,E1 -21916.863,E2 -21916.863} C_VEL
LIN {X 0,Y 192.608,Z 545.491,A -85,B 0,C 180,E1 -21921.663,E2 -21921.663} C_VEL
LIN {X 0,Y 192.596,Z 545.482,A -85,B 0,C 180,E1 -21926.815,E2 -21926.815} C_VEL
LIN {X 0,Y 192.66,Z 545.484,A -85,B 0,C 180,E1 -21931.692,E2 -21931.692} C_VEL
LIN {X 0,Y 192.68,Z 545.479,A -85,B 0,C 180,E1 -21936.346,E2 -21936.346} C_VEL
LIN {X 0,Y 192.726,Z 545.469,A -85,B 0,C 180,E1 -21941.46,E2 -21941.46} C_VEL
LIN {X 0,Y 192.758,Z 545.473,A -85,B 0,C 180,E1 -21945.214,E2 -21945.214} C_VEL
LIN {X 0,Y 192.977,Z 545.427,A -85,B 0,C 180,E1 -21949.509,E2 -21949.509} C_VEL
LIN {X 0,Y 193.058,Z 545.422,A -85,B 0,C 180,E1 -21951.628,E2 -21951.628} C_VEL
LIN {X 0,Y 193.26,Z 545.403,A -85,B 0,C 180,E1 -21957.917,E2 -21957.917} C_VEL
LIN {X 0,Y 193.442,Z 545.371,A -85,B 0,C 180,E1 -21960.001,E2 -21960.001} C_VEL
LIN {X 0,Y 192.99,Z 545.441,A -85,B 0,C 180,E1 -21964.178,E2 -21964.178} C_VEL
LIN {X 0,Y 193.038,Z 545.43,A -85,B 0,C 180,E1 -21968.375,E2 -21968.375} C_VEL
LIN {X 0,Y 192.799,Z 545.466,A -85,B 0,C 180,E1 -21972.635,E2 -21972.635} C_VEL
LIN {X 0,Y 192.755,Z 545.467,A -85,B 0,C 180,E1 -21976.96,E2 -21976.96} C_VEL
LIN {X 0,Y 192.634,Z 545.49,A -85,B 0,C 180,E1 -21981.399,E2 -21981.399} C_VEL
LIN {X 0,Y 192.662,Z 545.478,A -85,B 0,C 180,E1 -21984.226,E2 -21984.226} C_VEL
LIN {X 0,Y 192.649,Z 545.486,A -85,B 0,C 180,E1 -21988.893,E2 -21988.893} C_VEL
LIN {X 0,Y 192.599,Z 545.493,A -85,B 0,C 180,E1 -21993.187,E2 -21993.187} C_VEL
LIN {X 0,Y 192.608,Z 545.492,A -85,B 0,C 180,E1 -21996.609,E2 -21996.609} C_VEL
LIN {X 0,Y 192.534,Z 545.501,A -85,B 0,C 180,E1 -22001.076,E2 -22001.076} C_VEL
LIN {X 0,Y 192.699,Z 545.599,A -85,B 0,C 180,E1 -22006.496,E2 -22006.496} C_VEL
LIN {X 0,Y 194.947,Z 555.3,A -85,B 0,C 180,E1 -22011.413,E2 -22011.413} C_VEL
LIN {X 0,Y 195.225,Z 556.511,A -85,B 0,C 180,E1 -22011.972,E2 -22011.972} C_VEL
LIN {X 0,Y 204.336,Z 579.526,A -85,B 0,C 180,E1 -22014.462,E2 -22014.462} C_VEL
LIN {X 0,Y 206.911,Z 586.79,A -85,B 0,C 180,E1 -22015.151,E2 -22015.151} C_VEL
LIN {X 0,Y 210.389,Z 619.013,A -85,B 0,C 180,E1 -22017.017,E2 -22017.017} C_VEL
LIN {X 0,Y 209.403,Z 624.833,A -85,B 0,C 180,E1 -22017.137,E2 -22017.137} C_VEL
LIN {X 0,Y 203.376,Z 643.727,A -85,B 0,C 180,E1 -22017.172,E2 -22017.172} C_VEL
LIN {X 0,Y 202.479,Z 649.546,A -85,B 0,C 180,E1 -22017.312,E2 -22017.312} C_VEL
LIN {X 0,Y 201.373,Z 668.397,A -85,B 0,C 180,E1 -22018.113,E2 -22018.113} C_VEL
LIN {X 0,Y 200.076,Z 680.405,A -85,B 0,C 180,E1 -22018.942,E2 -22018.942} C_VEL
LIN {X 0,Y 198.303,Z 692.293,A -85,B 0,C 180,E1 -22020.108,E2 -22020.108} C_VEL
LIN {X 0,Y 196.411,Z 702.371,A -85,B 0,C 180,E1 -22021.408,E2 -22021.408} C_VEL
LIN {X 0,Y 193.964,Z 714,A -85,B 0,C 180,E1 -22023.36,E2 -22023.36} C_VEL
LIN {X 0,Y 191.505,Z 724.51,A -85,B 0,C 180,E1 -22025.616,E2 -22025.616} C_VEL
LIN {X 0,Y 189.255,Z 733.994,A -85,B 0,C 180,E1 -22028.202,E2 -22028.202} C_VEL
LIN {X 0,Y 187.745,Z 740.334,A -85,B 0,C 180,E1 -22030.312,E2 -22030.312} C_VEL
LIN {X 0,Y 185.901,Z 748.231,A -85,B 0,C 180,E1 -22033.529,E2 -22033.529} C_VEL
LIN {X 0,Y 184.493,Z 754.511,A -85,B 0,C 180,E1 -22036.788,E2 -22036.788} C_VEL
LIN {X 0,Y 183.74,Z 759.483,A -85,B 0,C 180,E1 -22040.089,E2 -22040.089} C_VEL
LIN {X 0,Y 183.425,Z 763.27,A -85,B 0,C 180,E1 -22043.4,E2 -22043.4} C_VEL
LIN {X 0,Y 183.453,Z 765.201,A -85,B 0,C 180,E1 -22045.606,E2 -22045.606} C_VEL
LIN {X 0,Y 183.527,Z 766.673,A -85,B 0,C 180,E1 -22047.805,E2 -22047.805} C_VEL
LIN {X 0,Y 183.573,Z 767.663,A -85,B 0,C 180,E1 -22050,E2 -22050} C_VEL
LIN {X 0,Y 183.442,Z 768.227,A -85,B 0,C 180,E1 -22052.196,E2 -22052.196} C_VEL
LIN {X 0,Y 183.271,Z 768.384,A -85,B 0,C 180,E1 -22054.399,E2 -22054.399} C_VEL
LIN {X 0,Y 183.251,Z 768.145,A -85,B 0,C 180,E1 -22056.607,E2 -22056.607} C_VEL
LIN {X 0,Y 183.47,Z 767.479,A -85,B 0,C 180,E1 -22058.814,E2 -22058.814} C_VEL
LIN {X 0,Y 184.503,Z 764.983,A -85,B 0,C 180,E1 -22063.211,E2 -22063.211} C_VEL
LIN {X 0,Y 186.033,Z 762.034,A -85,B 0,C 180,E1 -22066.459,E2 -22066.459} C_VEL
LIN {X 0,Y 188.157,Z 758.089,A -85,B 0,C 180,E1 -22069.643,E2 -22069.643} C_VEL
LIN {X 0,Y 191.27,Z 752.456,A -85,B 0,C 180,E1 -22073.059,E2 -22073.059} C_VEL
LIN {X 0,Y 194.702,Z 745.628,A -85,B 0,C 180,E1 -22076.242,E2 -22076.242} C_VEL
LIN {X 0,Y 198.676,Z 737.615,A -85,B 0,C 180,E1 -22079.103,E2 -22079.103} C_VEL
LIN {X 0,Y 202.491,Z 729.53,A -85,B 0,C 180,E1 -22081.373,E2 -22081.373} C_VEL
LIN {X 0,Y 206.969,Z 718.706,A -85,B 0,C 180,E1 -22083.782,E2 -22083.782} C_VEL
LIN {X 0,Y 211.062,Z 707.583,A -85,B 0,C 180,E1 -22085.641,E2 -22085.641} C_VEL
LIN {X 0,Y 214.384,Z 696.852,A -85,B 0,C 180,E1 -22087.039,E2 -22087.039} C_VEL
LIN {X 0,Y 217.465,Z 685.158,A -85,B 0,C 180,E1 -22088.175,E2 -22088.175} C_VEL
LIN {X 0,Y 220.103,Z 671.986,A -85,B 0,C 180,E1 -22089.095,E2 -22089.095} C_VEL
LIN {X 0,Y 221.813,Z 657.739,A -85,B 0,C 180,E1 -22089.777,E2 -22089.777} C_VEL
LIN {X 0,Y 224.387,Z 623.825,A -85,B 0,C 180,E1 -22090.963,E2 -22090.963} C_VEL
LIN {X 0,Y 223.695,Z 611.913,A -85,B 0,C 180,E1 -22091.891,E2 -22091.891} C_VEL
LIN {X 0,Y 220.341,Z 603.005,A -85,B 0,C 180,E1 -22093.575,E2 -22093.575} C_VEL
LIN {X 0,Y 216.364,Z 594.148,A -85,B 0,C 180,E1 -22095.689,E2 -22095.689} C_VEL
LIN {X 0,Y 212.656,Z 586.765,A -85,B 0,C 180,E1 -22097.815,E2 -22097.815} C_VEL
LIN {X 0,Y 209.414,Z 581.016,A -85,B 0,C 180,E1 -22099.873,E2 -22099.873} C_VEL
LIN {X 0,Y 206.44,Z 575.927,A -85,B 0,C 180,E1 -22101.975,E2 -22101.975} C_VEL
LIN {X 0,Y 203.175,Z 570.532,A -85,B 0,C 180,E1 -22104.633,E2 -22104.633} C_VEL
LIN {X 0,Y 198.039,Z 562.699,A -85,B 0,C 180,E1 -22110.208,E2 -22110.208} C_VEL
LIN {X 0,Y 194.836,Z 558.526,A -85,B 0,C 180,E1 -22116.108,E2 -22116.108} C_VEL
LIN {X 0,Y 194.142,Z 557.099,A -85,B 0,C 180,E1 -22119.366,E2 -22119.366} C_VEL
LIN {X 0,Y 194.269,Z 557.087,A -85,B 0,C 180,E1 -22124.256,E2 -22124.256} C_VEL
LIN {X 0,Y 197.155,Z 558.484,A -85,B 0,C 180,E1 -22130.862,E2 -22130.862} C_VEL
LIN {X 0,Y 198.429,Z 561.358,A -85,B 0,C 180,E1 -22132.942,E2 -22132.942} C_VEL
LIN {X 0,Y 200.685,Z 563.574,A -85,B 0,C 180,E1 -22135.48,E2 -22135.48} C_VEL
LIN {X 0,Y 201.906,Z 564.366,A -85,B 0,C 180,E1 -22136.603,E2 -22136.603} C_VEL
LIN {X 0,Y 204.069,Z 567.633,A -85,B 0,C 180,E1 -22138.615,E2 -22138.615} C_VEL
LIN {X 0,Y 205.378,Z 569.116,A -85,B 0,C 180,E1 -22139.631,E2 -22139.631} C_VEL
LIN {X 0,Y 207.73,Z 572.801,A -85,B 0,C 180,E1 -22141.431,E2 -22141.431} C_VEL
LIN {X 0,Y 209.158,Z 574.575,A -85,B 0,C 180,E1 -22142.392,E2 -22142.392} C_VEL
LIN {X 0,Y 212.463,Z 579.321,A -85,B 0,C 180,E1 -22144.446,E2 -22144.446} C_VEL
LIN {X 0,Y 216.957,Z 586.457,A -85,B 0,C 180,E1 -22146.955,E2 -22146.955} C_VEL
LIN {X 0,Y 221.706,Z 594.69,A -85,B 0,C 180,E1 -22149.328,E2 -22149.328} C_VEL
LIN {X 0,Y 225.844,Z 602.901,A -85,B 0,C 180,E1 -22151.21,E2 -22151.21} C_VEL
LIN {X 0,Y 222.242,Z 647.583,A -85,B 0,C 180,E1 -22152.788,E2 -22152.788} C_VEL
LIN {X 0,Y 220.362,Z 661.044,A -85,B 0,C 180,E1 -22153.603,E2 -22153.603} C_VEL
LIN {X 0,Y 217.986,Z 673.391,A -85,B 0,C 180,E1 -22154.717,E2 -22154.717} C_VEL
LIN {X 0,Y 214.936,Z 685.357,A -85,B 0,C 180,E1 -22156.161,E2 -22156.161} C_VEL
LIN {X 0,Y 211.463,Z 696.329,A -85,B 0,C 180,E1 -22157.867,E2 -22157.867} C_VEL
LIN {X 0,Y 207.526,Z 706.811,A -85,B 0,C 180,E1 -22159.974,E2 -22159.974} C_VEL
LIN {X 0,Y 203.276,Z 716.615,A -85,B 0,C 180,E1 -22162.529,E2 -22162.529} C_VEL
LIN {X 0,Y 199.585,Z 724.079,A -85,B 0,C 180,E1 -22164.995,E2 -22164.995} C_VEL
LIN {X 0,Y 195.983,Z 730.732,A -85,B 0,C 180,E1 -22167.786,E2 -22167.786} C_VEL
LIN {X 0,Y 192.896,Z 736.071,A -85,B 0,C 180,E1 -22170.668,E2 -22170.668} C_VEL
LIN {X 0,Y 190.207,Z 740.341,A -85,B 0,C 180,E1 -22173.657,E2 -22173.657} C_VEL
LIN {X 0,Y 187.956,Z 743.613,A -85,B 0,C 180,E1 -22176.745,E2 -22176.745} C_VEL
LIN {X 0,Y 185.703,Z 746.435,A -85,B 0,C 180,E1 -22180.809,E2 -22180.809} C_VEL
LIN {X 0,Y 184.615,Z 747.542,A -85,B 0,C 180,E1 -22183.674,E2 -22183.674} C_VEL
LIN {X 0,Y 183.78,Z 747.927,A -85,B 0,C 180,E1 -22186.599,E2 -22186.599} C_VEL
LIN {X 0,Y 183.205,Z 747.486,A -85,B 0,C 180,E1 -22190.104,E2 -22190.104} C_VEL
LIN {X 0,Y 183.091,Z 745.97,A -85,B 0,C 180,E1 -22193.714,E2 -22193.714} C_VEL
LIN {X 0,Y 183.555,Z 743.11,A -85,B 0,C 180,E1 -22197.587,E2 -22197.587} C_VEL
LIN {X 0,Y 184.399,Z 739.119,A -85,B 0,C 180,E1 -22201.232,E2 -22201.232} C_VEL
LIN {X 0,Y 185.363,Z 734.924,A -85,B 0,C 180,E1 -22204.135,E2 -22204.135} C_VEL
LIN {X 0,Y 186.725,Z 729.155,A -85,B 0,C 180,E1 -22207.308,E2 -22207.308} C_VEL
LIN {X 0,Y 188.566,Z 722.029,A -85,B 0,C 180,E1 -22210.401,E2 -22210.401} C_VEL
LIN {X 0,Y 190.693,Z 713.433,A -85,B 0,C 180,E1 -22213.378,E2 -22213.378} C_VEL
LIN {X 0,Y 192.991,Z 703.797,A -85,B 0,C 180,E1 -22216.04,E2 -22216.04} C_VEL
LIN {X 0,Y 195.308,Z 693.303,A -85,B 0,C 180,E1 -22218.322,E2 -22218.322} C_VEL
LIN {X 0,Y 197.425,Z 682.342,A -85,B 0,C 180,E1 -22220.209,E2 -22220.209} C_VEL
LIN {X 0,Y 199.17,Z 671.599,A -85,B 0,C 180,E1 -22221.664,E2 -22221.664} C_VEL
LIN {X 0,Y 200.817,Z 658.857,A -85,B 0,C 180,E1 -22222.964,E2 -22222.964} C_VEL
LIN {X 0,Y 202.008,Z 645.664,A -85,B 0,C 180,E1 -22223.884,E2 -22223.884} C_VEL
LIN {X 0,Y 203.317,Z 622.618,A -85,B 0,C 180,E1 -22224.816,E2 -22224.816} C_VEL
LIN {X 0,Y 205.074,Z 587.183,A -85,B 0,C 180,E1 -22226.138,E2 -22226.138} C_VEL
LIN {X 0,Y 198.168,Z 570.973,A -85,B 0,C 180,E1 -22227.912,E2 -22227.912} C_VEL
LIN {X 0,Y 187.869,Z 549.876,A -85,B 0,C 180,E1 -22230.675,E2 -22230.675} C_VEL
LIN {X 0,Y 186.491,Z 547.318,A -85,B 0,C 180,E1 -22231.056,E2 -22231.056} C_VEL
LIN {X 0,Y 186.273,Z 546.283,A -85,B 0,C 180,E1 -22231.165,E2 -22231.165} C_VEL
LIN {X 0,Y 185.967,Z 546.32,A -85,B 0,C 180,E1 -22236.51,E2 -22236.51} C_VEL
LIN {X 0,Y 185.94,Z 546.323,A -85,B 0,C 180,E1 -22240.672,E2 -22240.672} C_VEL
LIN {X 0,Y 185.722,Z 546.349,A -85,B 0,C 180,E1 -22245.36,E2 -22245.36} C_VEL
LIN {X 0,Y 185.604,Z 546.36,A -85,B 0,C 180,E1 -22249.924,E2 -22249.924} C_VEL
LIN {X 0,Y 185.598,Z 546.365,A -85,B 0,C 180,E1 -22254.662,E2 -22254.662} C_VEL
LIN {X 0,Y 185.576,Z 546.367,A -85,B 0,C 180,E1 -22259.493,E2 -22259.493} C_VEL
